# B&R Automation Studio project NewPendant_NG4_11_05_25A (part 6)

#### Main2_FourAxisTigCtrl.c.c
```c
/********************************************************************
 * COPYRIGHT -- wsi
 ********************************************************************
 * Program: Master
 * File: Master.c
 * Author: wsi
 * Created: September 25, 2012
 ********************************************************************

 Hardware[1].Inp[23] - index 80x switch
 * Implementation of program Master
 ********************************************************************/
#include <bur/plctypes.h>

#ifdef _DEFAULT_INCLUDES
#include <AsDefault.h>
#endif

#include <math.h>

#include <..\GlobDef.h>
#include <..\..\Lib\WSI_Lib.c>

#include <..\GlobDecl.h>
#include <..\Hardcoded.c>
#include <..\HMI_Cntrl.c>
#include <..\HeadConfig.c>

#include <..\..\Lib\Statelib.c>
#include <..\..\Lib\LCDLib.c>
#include <..\..\Lib\DrillMenuLib.c>
#include <..\..\Lib\LoggerLib.c>

//#include <..\..\Lib\utilityLib\bgdebug.h>
//#define TEST_ONLY_PLC_ANDROID
#define HASH_NUM				442
//#define VERSION "UnivCntrl-10-29-19B" was tested by welders
//#define VERSION "UnivCntrl-11-20-19F" // was ready for testing before Thanksgiving but nobody tested it
//#define VERSION "UnivCntrl-01-10-20F" // Successfully tested in January - very good result
//#define VERSION "UnivCntrl-02-14-20F"
//#define VERSION "UnivCntrl-02-17-20B"
//#define VERSION "UnivCntrl-02-27-20B"
//#define VERSION "UnivCntrl-03-13-20Exp"
//#define VERSION "UnivCntrl-04-17-20A" // ESTOP does not interrupt GAS
//#define VERSION "UnivCntrl-05-15-20exp" // was working
//#define VERSION "UnivCntrl-06-12-20exp"  // Max Osc ampit was changed to 3 inch
// New OSC Concept for BPV v2 is possible - make changes in Configure_BPV_v2 in OSC motor def and OSC Process use type 10
//#define VERSION "UnivCntrl-06-16-20F"  //  New Heads: BPV 2.0 MT-BO (replaces "BPV 2.0 MPBO") , BPV 2.0 TT-BO , BPV 2.0 MT-BO_TOS , BPV 2.0 TT-BO_TOS;
//BPV_v2_TT_BO_TOS chyba dziala , przenioslem w desperacji wszystko z MBPOH , trzeba dodac w Main2 wszystko zwiazane z nowymi headami
//#define VERSION "UnivCntrl-07-10-20A"
//#define VERSION "UnivCntrl-07-23-20A"
//#define VERSION "UnivCntrl-07-27-20A"
//#define VERSION "UnivCntrl-08-20-20F" // good working install on 5 machines in October 2020
//#define VERSION "UnivCntrl-09-14-20B" // new TML organization )comments) - just started
//#define VERSION "UnivCntrl-09-16-20A" // new TML organization (comments) - compiled but never used
//#define VERSION "UnivCntrl-10-27-20A" // new TML organization (comments) + SweachtHead for WF is fixed in SuperMini- is tested
//#define VERSION "UnivCntrl-11-19-20F" // the exactly the same as  "UnivCntrl-10-27-20A" but installed on Tyler machine
//#define VERSION "UnivCntrl-11-24-20F" // all as above plus file name fixed
//#define VERSION "UnivCntrl-01-29-21F" // Installed on real machine with SMH

//#define VERSION "UnivCntrl-06-04-21B" // starting - adding weld report HMI

//#define VERSION "UnivCntrl-08-09-21G" // wyjechalo do Occonee - na razie spakowane - dzialalo dobrze byli zadowloeni
//#define VERSION "UnivCntrl-08-26-21A" // proba uzycia CMT

//#define VERSION "UnivCntrl-09-02-21A" // Mode 2 nie dzialal w SuperMini ?? spowrotem Mode 1 //TVL_ROT_Param_Set[i].Mode = 2; //TVL_MODE_BPV_PosMode
// aby dzialal TVL Mode 2,3 - jazda wg position to trzeba dodac w drivie POSTRIGG2=2147483647 , POSTRIGG3=2147483647 , POSTRIGG4=2147483647
//#define VERSION "UnivCntrl-09-21-21F"
//define VERSION "MIGE_EXP-10-11-21F"
//#define VERSION "MIGE_EXP-10-13-21F"
//#define VERSION "MIGE_EXP-10-14-21G"
//#define VERSION "MIGE_EXP-10-15-21F"
//#define VERSION "MIGE_EXP-10-19-21F"
//#define VERSION "UnivCntrl-10-19-21F"
//#define VERSION "UnivCntrl-10-19-21M"
//#define VERSION "UnivCntrl-10-19-21MX"
//#define VERSION "UnivCntrl-11-02-21MX"
//#define VERSION "UnivCntrl-11-10-21MX"  // Zmiany W MIG EXP - 0.5 s delay przy restarcie pojednyczych TML
//#define VERSION "UnivCntrl-11-10-21MX"  // Zmiany W MIG EXP - 0.5 s delay przy restarcie pojednyczych TML

//#define VERSION "UnivCntrl-02-16-22A"  // dziala RUBIX

//#define VERSION "UnivCntrl-02-23-22A"  // dzial  MINI Standard

//#define VERSION "UnivCntrl-03-01-22F"  // Synch Pulse  MINI Standard & Rubix

//#define VERSION "UnivCntrl-03-24-22F"  // Poprawki w beat logger + Synch Pulse  MINI Standard & Rubix

//#define VERSION "UnivCntrl-04-05-22F"  // MiniHead Omega  +>   Poprawki w beat logger + Synch Pulse  MINI Standard & Rubix
// required -> UnivCntrl_01Apr22_US_4AXIS RUBIX & STND&MiniOmega.m.zip

//#define VERSION "UnivCntrl-04-12-22H" // poprawiony TVL step w Mode 2 i 3
// required -> UnivCntrl_01Apr22_US_4AXIS RUBIX & STND&MiniOmega.m.zip

//#define VERSION "UnivCntrl-04-29-22F" // nowy D-Head
// required -> UnivCntrl_29Apr22_US_4AXIS RUBIX & STND&MiniOmega&DHead.m.zip

//#define VERSION "UnivCntrl-06-23-22F" // nowy D-Head
// required -> UnivCntrl_21June22_US_4AXIS RUBIX & STND&MiniOmega&DHead.m.zip

// this was changed TVL_ROT_Param_Set[i].Mode = 3; to Mode 1
// in BPV_v2_MPBO head to get infinity welding
//#define VERSION "UnivCntrl-12-05-23F"
// required -> UnivCntrl_21June22_US_4AXIS RUBIX & STND&MiniOmega&DHead.m.zip

// New Head definition - BPV v2 MT  - like BPV2 but with MT truck - no position mode in TVL
//#define VERSION "UnivCntrl-12-06-23F"
// required -> UnivCntrl_21June22_US_4AXIS RUBIX & STND&MiniOmega&DHead.m.zip

//#define VERSION "UnivCntrl-12-11-23F" //New Head definition - BPV v1 MT
// required -> UnvCntrl_BPV_11_12_23.m // nowy TVL head
// required -> UnivCntrl_21June22_US_4AXIS RUBIX & STND&MiniOmega&DHead.m.zip

//#define VERSION "UnivCntrl-12-14-23F" //WYWALONY potencjometr z AVC New Head definition - BPV v1 MT
// required -> UnvCntrl_BPV_11_12_23.m // nowy TVL head
// required -> UnivCntrl_21June22_US_4AXIS RUBIX & STND&MiniOmega&DHead.m.zip

//#define VERSION "UnivCntrl-07-12-24A" // dodane BPV_v2_Video i zmiany W HMI Report

//#define VERSION "UnivCntrl-07-23-24A" // dodane BPV_v2_Video i zmiany W HMI Report

//#define VERSION "UnivCntrl-07-31-24F" // all above plus AVC feedback calibration in all legacy heads fixed

//#define VERSION "UnivCntrl-08-01-24G" // Weld Report : Heat Input or Power Ratio

//#define VERSION "UnivCntrl-09-09-24G" // Weld Report : Heat Input or Power Ratio + Limits

//#define VERSION "UnivCntrl-09-09-24R" // Radom - Weld Report : Heat Input or Power Ratio + Limits

//#define VERSION "UnivCntrl-10-18-24A" // new head : ClamShell , small change in reports

//#define VERSION "UnivCntrl-11-07-24A" // New Head KKL
//#define VERSION "UnivCntrl-11-29-24A" // New Head KKL
//#define VERSION "UnivCntrl-12-02-24A" // New Head KKL
//#define VERSION "UnivCntrl-12-03-24A" // New Head KKL

//#define VERSION "UnivCntrl-12-04-24F" // taki zostawiam przed wyjazdem
//#define VERSION "UnivCntrl-12-11-24A" // Added cherrypoint head - BP

//#define VERSION "UnivCntrl-12-30-24A" // Wire Angle Btn Fixed

/*
#ifdef MIG_SYSTEM
	#define VERSION "NG4_C15-01-14-25A" // Wire Angle Zero Btn Fixed
#else
	#ifdef CMT_SYSTEM
		#define VERSION "CMT_C15-01-14-25A"
	#else
		#define VERSION "MPC_C15-01-14-25A" // Wire Angle Zero Btn Fixed
	#endif
#endif*/

//#define VERSION "01-16-25H"  // Universal version for ClamSHell , CherryPoint & CMT , New Weld Report

//#define VERSION "01-27-25A"  // Weld Report changes - new drives cfg for ClamShell
// required -> UnvCntrl_CLAMSHELL_2025_27Jan.m

//#define VERSION "01-30-25F"  // One Wrist for BPV video Weld Report changes - new drives cfg for ClamShell ,
// required -> UnvCntrl_CLAMSHELL_2025_27Jan.m

//#define VERSION "02-03-25A"  // new head - Cherry Point BPV2 Mig Track, ++ w TVL_ROT gdy TVL continues zmiana na Mode 1
// required -> UnvCntrl_CLAMSHELL_2025_27Jan.m

//#define VERSION "02-12-25F"  // WRST TML calling fixed TML_mgr[0].hrdw[1].AxisNum = 13;
// required -> UnvCntrl_CLAMSHELL_2025_27Jan.m
//#define VERSION "02-13-25F"  // Limited list of heads
//#define VERSION "02-18-25F"  // Problem with TVL MT Mode 3 solved - Limited list of heads

// Nowy runtime , Nowe App_Config_ID i inaczej pamiec skonfigurowana
//#define VERSION "03-11-25A"  // WF & WP dziala
//#define VERSION "03-12-25A"  // AVC sense dziala
//#define VERSION "03-13-25F"  // To dzialalo i spawalo

//#define VERSION "03-13-25K"  // dodano klucz NG4_TIG_SYSTEM
//required -> UnvCntrl_CLAMSHELL_2025_27Jan.m
// required -> UnvCntrl_MIG_TIG_13Mar2025

//#define VERSION "08-01-25A"  // Nowy Pendant NG4 - proba na maszynie

//#define VERSION "08-06-25J"  // Nowy Pendant NG4 ale proba na maszynie NG4 controler

//#define VERSION "08-07-25A"  // Nowy Pendant NG4 ale proba na maszynie NG4 controler
//#define VERSION "08-07-25K"  // Nowy Pendant NG4 proba na maszynie NG4 controler _PODSTAWA do Krakowa - SPAWAL

//#define VERSION "08-11-25B"  // base for VNC pendant development

//#define VERSION "09-01-25A" // pierwsze prace w Krakowie
//#define VERSION "09-02-25A" // pierwsze prace w Krakowie
//#define VERSION "09-03-25B" // pierwsze prace w Krakowie

//#define VERSION "09-05-25A" // pierwsze prace w Krakowie
//#define VERSION "09-06-25A" // pierwsze prace w Krakowie

//#define VERSION "09-08-25A" // pierwsze prace w Krakowie
//#define VERSION "09-11-25A" // pierwsze prace w Krakowie

//#define VERSION "09-12-25A" // pierwsze prace w Krakowie

//#define VERSION "09-14-25A" // pierwsze prace w Krakowie

//#define VERSION "09-16-25A" // pierwsze prace w Krakowie
//#define VERSION "09-17-25A" // pierwsze prace w Krakowie
//#define VERSION "09-18-25A" // pierwsze prace w Krakowie
//#define VERSION "09-19-25A" // Taki przylecial z Krakowa

//#define VERSION "10-21_25A" // pierwsze uruchomienie na maszynie
//#define VERSION "10-22_25A" // proba uruchomienia tez na MPC
//#define VERSION "10-24_25D" // proba uruchomienia tez na MPC
//#define VERSION "10-30_25B" // start na CLAM SHELL maszynie
//#define VERSION "10-31_25D" // start na CLAM SHELL maszynie

//#define VERSION "11-03_25A" // start na CLAM SHELL maszynie
//#define VERSION "11-04_25A" // start na CLAM SHELL maszynie

#define VERSION "11-05_25A" // TVL Balance DIst. added

// For new pendant
_GLOBAL HARDWARE_obj hardware;
_GLOBAL MTR_obj motors[4]; // NUM_MOTORS

void FourAxisTIG();

/////////////////

_LOCAL DINT 	statusInit;

_LOCAL plcbit   MIG_ESTOP_Rst_Out , MIG_ESTOP_Rst_Btn_Inp , MIG_ESTOP_Rst_PendantBtn;

_LOCAL Cfg_typ *cfg;
_LOCAL CurCfg_typ *curCfg;
_LOCAL CurCalib_typ *curCalib, *defCalib;
_LOCAL Scaled_Var_obj *var;

_LOCAL MASTER_typ * m;
_LOCAL SerialPortDriver_typ * rs;
_LOCAL LCD_MGR_obj * lcd;
_LOCAL PENDANT_HARDWARE_obj * pend;
_LOCAL HMI_typ * hmi;
_LOCAL HMI_INTRF_typ * intrf;

_LOCAL LCD_NODE_obj * nodes;
_LOCAL TON_typ	WF_Catch_TMR;
_LOCAL UINT 	WF_RAMPUP_Comp_Step;

_LOCAL TON_typ	DoubleStop_TMR;
_LOCAL plcbit	DoubleStopBtn;
_LOCAL plcbit	DoubleStopBtn_Latch, StopBtn_Latch;

_LOCAL TON_typ	ESTOP_Dly_Tmr, AndroidConnect_Tmr;
_LOCAL UDINT	GlblBtnLED_Mask;
_LOCAL plcbit	ESTOP_PERMIT;

_LOCAL TON_typ Restart_Tmr;

//_LOCAL UINT CalibStep;
//_LOCAL BOOL CalibStepDone;
prcsSTATUS_Enum _ProcStatus;

_LOCAL INT		ANDROID_Pendant;
_LOCAL plcbit	StartBtn, StopBtn;

_LOCAL TON_typ	WireDisable_TMR;
_LOCAL UINT 	TVL_Latch_Cnt, TVL_Latch_Tm;
_LOCAL UINT 	TVL_Latch_Latched, _TVL_Latch_Latched;

_LOCAL plcbit   SYSTEM_LOCKED;

_LOCAL plcbit	Force_ENTR_LCD, _Force_ENTR_LCD;
_LOCAL UINT 	DebaunceCnt[16], DebounceTickSw, DebounceTickSwMax;
_LOCAL BOOL 	TickSw, _TickSw;
_LOCAL DINT 	WF_TVL_Diff;

INT 			_curZone;

_LOCAL plcbit	FirstScan, RefreshAndroid;

_LOCAL DINT 	_TIG_Mode , _AVC_Mode , _TVL_SYN_MODE , _WF_SYN_MODE , _WP_SYN_MODE ;

BOOL			SendRS232, _SendRS232;
_LOCAL plcstring txt[16][32];
_LOCAL Calib_Param_typ tempCalib;

_LOCAL plcbit	_segmSw;

_LOCAL plcbit	ROM_USB;

//_LOCAL DINT 	_SETUP_HEAD_SETUP;
_LOCAL plcbit	AutoStartEnable;

_LOCAL DINT 	actTicks, actTickBalance, actRot, _actRot, actPathCnt;
_LOCAL DINT 	deltaTick, actTicksForZone, actTicksForHead, actTVL_Dist, encHome_TVL;
_LOCAL DINT 	tickEncoder, _tickEncoder, encDelta;
_LOCAL UINT 	btnProgress, btnProgressMax, btnProgressBias;
_GLOBAL UINT 	curTML_indx , TML_Setup_From_Diagn;
_LOCAL UINT	    stillRun;

float			_TIG_CalibAmp, _HW_CalibAmp;

//_LOCAL Calib_Param_typ tempCalibPar;
_LOCAL UINT			_ToolHeadID , _ToolHeadID_Sw1 , _ToolHeadID_Sw2;
DINT			_GlblBtnCmd[2];

INT 			_AndroidWheel;
UINT			_AndroidEntrBtn;
_LOCAL plcstring LineTxt[256];
_LOCAL INT		parametersDump_Step, paramIndx;
_LOCAL DTStructure DTStruct;
_LOCAL DTGetTime_typ DTGetTime_1;

UDINT			_datagramCountTotal[2];
UDINT			_datagramPerSec[2];

USINT 			_MappingActive;

UINT			_PLC_Changes;
USINT 			_WireDisabled;
_LOCAL plcbit	AutoStartBtn;
_LOCAL plcbit	Cont_Stop_By_End;

_LOCAL plcbit   TIG_MIG_Sw_Inp;

_LOCAL plcbit   MIG_ESTOP_Rst_Out , MIG_ESTOP_Rst_Btn_Inp, MIG_ESTOP_Rst_Btn_Virt;
_LOCAL plcbit   Pend_Btn_Start_Virt , Pend_Btn_Stop_Virt;
_LOCAL plcbit 	MIG_Btn_Left_Inp, MIG_Btn_Right_Inp , MIG_Btn_Stop_Inp;

_LOCAL plcbit 	MIG_Btn_Left_Inp_Virt, MIG_Btn_Right_Inp_Virt ;

//_LOCAL UINT POPUP_EVENT;

_LOCAL plcbit ESTOP_Inp_Status;

_LOCAL Robot_typ * robot;

_LOCAL UINT KK_ErrorsHold;
_LOCAL UINT KK_Can_Download_Everything;

_LOCAL USINT KK_Was_Cahnged , KK_Catched;
_LOCAL USINT	KK_Life;
_LOCAL BOOL 	KK_AUTO_Test;
_LOCAL plcstring KK_text[64];
_LOCAL INT		KK_AndroidWheelIncr;
_LOCAL INT		KK_Drill, KK_Out, KK_ZONE;
_LOCAL DINT 	KK_actPosProcss , KK_ActEnc;
_LOCAL float	KK_CatchAndroidComErr;
_LOCAL UINT 	KK_CatchAndroidErr;
_LOCAL UINT 	KK_test;
_LOCAL plcbit 	KK_ClearErr;

_LOCAL USINT KK_FirstRestart_Loop;

_LOCAL DINT 	myCounter;

_LOCAL USINT   AmpsCalib_step;

_LOCAL UINT TML_Restart_Indx , TML_Restart_Step;
_LOCAL UINT Process_Restart_Indx , Process_Restart_Step;

_LOCAL float KK_ZigZag_Dist , KK_Balance_Dist;

// TVL_MAPPing
_GLOBAL DINT _deltaAPOS[TML_SERVO_NUM] , _deltaAPOS2[TML_SERVO_NUM];
_GLOBAL UINT TVL_MAP_Indx[TML_SERVO_NUM], TVL_MAP_Indx_New[TML_SERVO_NUM];
_LOCAL  UINT TVL_MAP_Step;
_LOCAL  plcbit TVL_MAP_Allowed;
void TVL_Map_ToFile();

void ProcessEvents_Android(MASTER_typ * m, LCD_NODE_obj * nodes, HMI_typ * hmi, HMI_INTRF_typ * intrf);
void EditParam(UINT paramIndx);
void JogProcessAndroid(HMI_INTRF_typ * intrf, UINT procIndx, float gain);
void TakeNextWeldProgram(HMI_typ * hmi);
void AndroidHelper(MASTER_typ * m, UINT n);

void CalibrationModePendantButtons(MASTER_typ * m, HMI_typ * hmi, HMI_INTRF_typ * intrf, LCD_MGR_obj * lcd);
void StopModeAndroidButtons(MASTER_typ * m, HMI_typ * hmi, HMI_INTRF_typ * intrf, LCD_MGR_obj * lcd);
void StopCalibrationModeAndroidButtons(MASTER_typ * m, HMI_typ * hmi, HMI_INTRF_typ * intrf, LCD_MGR_obj * lcd);
void RunModeAndroidButtons(MASTER_typ * m, HMI_typ * hmi, HMI_INTRF_typ * intrf, LCD_MGR_obj * lcd);
void RunCalibrationModeAndroidButtons(MASTER_typ * m, HMI_typ * hmi, HMI_INTRF_typ * intrf, LCD_MGR_obj * lcd);

DINT MasterSequence(MASTER_typ * m, HMI_typ * hmi, plcbit StartBtn, plcbit StopBtn);
DINT MasterSequence_Contin(MASTER_typ * m, HMI_typ * hmi, plcbit StartBtn, plcbit StopBtn);
DINT MasterSequence_Contin_OneWay(MASTER_typ * m, HMI_typ * hmi, plcbit StartBtn, plcbit StopBtn);

DINT CalibrationSequence(MASTER_typ * m, HMI_typ * hmi, plcbit StartBtn, plcbit StopBtn);

void IncrParam(CurCfg_typ * curCfg, UINT param, DINT segm, float gain);
void DecrParam(CurCfg_typ * curCfg, UINT param, DINT segm, float gain);

void Check_parOSC_Excur(CurCfg_typ * curCfg, HMI_typ * hmi, UINT seg);

void Check_parOSC_Amplit(CurCfg_typ * curCfg, HMI_typ * hmi, UINT seg);
void PleaseUpdateHeadSetup(MASTER_typ * m);

void SetBannerTxt(MASTER_typ * m, HMI_typ * hmi, HMI_INTRF_typ * intrf);
float getBtnProgress();
void SetZeroPosition(MASTER_typ * m);
void CreateParamList();
void DeleteExtension(char * p);
void WireDisableInable(plcbit Tmr_Q);

void DumpParamToFile();
void EvaluatePosition();
void Fill_Segments(CurCfg_typ * curCfg, UINT par, UINT seg, UINT Mode, UINT Step);

int WatchArcLinkError(MASTER_typ * m, Robot_typ * robot);
DINT Check_OSC_Amplt_and_Center();

void CalculateRunOverlap();
void CalculateRunOverlap_Cont();
void CalculateRunOverlap_Cont_OneWay();

void RestartStateMach();
plcbit Find_ext_txt(char *name , char* ext);

_LOCAL DINT _NextHeadConfig_Indx;

void _INIT Main2_INIT(void)
{
UINT i;

	KK_ZigZag_Dist = 20;

	//////////////////////////////////
		// Pozostalosci po SuperMaster
		// do przeanalizowania
	#ifdef  MIG_SYSTEM

		ProjectConfig_Hrdw = project_FourAxisTig;
		ProjectConfig = project_FourAxisTig;

	#endif
		FourAxisTIG();

	///////////////////////////////////

#ifdef MIG_SYSTEM
	strcpy(PLC_Version_TXT, "NG4-"); //#define VERSION "NG4_C15-01-14-25A" // Wire Angle Zero Btn Fixed
#else
	#ifdef CMT_SYSTEM
	strcpy(PLC_Version_TXT, "CMT-");
	#else
	strcpy(PLC_Version_TXT, "MPC-");
	#endif
#endif

	strcat(PLC_Version_TXT, VERSION);

#ifdef CHERRYPOINT_LIST

	strcat(PLC_Version_TXT, "-CP");

#endif

	LimScal_Tilt.x1 = 0.0;
	LimScal_Tilt.y1 = 0.0;

	LimScal_Tilt.x1 = 4096.0;
	LimScal_Tilt.y1 = 360.0;

	//	Program options
	KK_DoNotChangeTMLProgram 	= 0;
	KK_DoNotHashCalculation 	= 1; // always like that
	TVL_MAP_Allowed 			= 0;
	KK_No_TVL_Restart	= 0;
	KK_ManualCalib		= 0;
	KK_TML_PowerON		= 0;
	KK_Functionality	= 0;
	KK_ErrorsHold 		= 0;
	KK_Can_Download_Everything = 0;

	//////////////////////////
	Hold_Estop_ON 		= 0;
	ESTOP_Inp_Status 	= 0;
	TVL_Latch_Tm		= 50;
	ANDROID_Pendant 	= 1;

	//some heads setup in Config
	btnProgressMax		= 50;
	btnProgressBias 	= 10;

	KK_AUTO_Test		= 0;

	DebounceTickSwMax	= 2;

	// Just to see globals in the watch window
	Master[0].Active	= Master[0].Active;

	//LCD_MGR[0].curHead = LCD_MGR[0].curHead;
	RS232[0].Ident		= RS232[0].Ident;
	Pendant[0].ABEncoder = Pendant[0].ABEncoder;

	ESTOP_Dly_Tmr.PT	= 1000; 					// 1 sec delay off ESTOP
	Hardware[0].Inp[4]	= 1;						// ESTOP

	Master[0].AndIntrf[0].Alive = 0;

	myCounter			= myCounter;

	ReadPermMemory_HS.Go = 0;
	ReadPermMemory_HS.Ready = 0;

	ReadCfgFile_HS.Go = 0;
	ReadCfgFile_HS.Ready = 0;

	TimerStart(&DoubleStop_TMR, 1.0);
	TimerExecute(&DoubleStop_TMR);

	Hardware[1].Outp[9] = 0; // Lights OFF (NC) on camera

	FirstScan = 1;
	RefreshAndroid = 0;

	SYSTEM_LOCKED = 0;

	LoggerInit(&LogMgr, &LogID, "LogBook1", 2000);

	// Very Important - get value from Statis Memory
	_NextHeadConfig_Indx = NextHeadConfig_Indx;
	actTicks			= actTicksPerm;

	if((_NextHeadConfig_Indx < 0) || (_NextHeadConfig_Indx >= HEAD_INVALID)){
		_NextHeadConfig_Indx = BPV_v2;
		NextHeadConfig_Indx = BPV_v2;
	}

	Master[0].ToolHeadID = (UINT)LastHeadDir;

	for(i = 0; i < HEAD_INVALID ; i++)
		AssignHeadText(NewHeadName[i] , i);

	strcpy(curHeadName , NewHeadName[NextHeadConfig_Indx]);

}

void _CYCLIC Main2_CYCLIC(void)
{
int 			i, k;
char			status, _status;
DINT			d;
int 			len;
float 			x;

//plcbit StartBtn , StopBtn;
INT 			tickIncr;
LCD_NODE_obj *	curNode;

	#ifdef MIG_PENDANT

		m		= pMaster[1];
		lcd 	= pLCD_MGR[1];
		rs		= pRS232[1];
		pend	= pPendant[1];

	#else

		m		= pMaster[0];
		lcd 	= pLCD_MGR[0];
		rs		= pRS232[0];
		pend	= pPendant[0];

	#endif

	if(SYSTEM_LOCKED) // System Locked after Head definition changed - Must reboot
		return;

	// Check if pointers are not null
	if (!m)
		return;

	nodes				= m->pNode[0];

	if (!nodes)
		return;

	if (!lcd)
		return;

	if (!rs)
		return;

	if (!pend)
		return;

	if (!m->pCurCfg || !m->pCfg || !m->pCalib || !m->pScaledVar)
		return;

	cfg 				= (Cfg_typ *)		m->pCfg;
	curCfg				= (CurCfg_typ *)	m->pCurCfg;
	curCalib			= (CurCalib_typ *)	m->pCalib;
	defCalib			= (CurCalib_typ *)	m->pDefaultCalib;
	var 				= (Scaled_Var_obj*)	m->pScaledVar;
	robot				= (Robot_typ*)PS_Param_Set[0].pArcLinkRobot;

	hmi 				= &m->Hmi[0];
	intrf				= &m->Intrf[0];

	if (!hmi || !intrf)
		return;

	////////////////////////////////////////

	if(KK_ClearErr){
		KK_ClearErr = 0;
		KK_AckAllErrors(&ErrorMgr);
	}
	//////////////////////////////////////

	Hardware[1].Outp[8] = Hardware[1].Outp[9]; // Power on Camera #1

	///////// Important because HMI in Global setting can change NextHeadConfig_Indx

	// Head type was changed - Load New Head definition

	if(hmi->curHeadID != P_PARAM_GLOBAL){

		if(_NextHeadConfig_Indx != NextHeadConfig_Indx){
			_NextHeadConfig_Indx = NextHeadConfig_Indx;

			LogTxt(&LogMgr, "Head was changed");

			/*
			STOP_SavingData = 1;
			m->sm.Step = 1001;
			m->LOCKED = 1;
			TML_MTR_CUT_POWER = 1;
			*/

			FirstScan = 1;

			#ifdef  MIG_PENDANT

			m->sm.Step = 1;

			#else

			RefreshAndroid = 1;
			TML_MTR_CUT_POWER = 1;

			m->LOCKED = 1;
			m->sm.Step = 250;

			#endif

		}

	}

	if(FirstScan){
		FirstScan = 0;

		ReadPermMemory_HS.Ready = 0;
		ReadPermMemory_HS.Go = 1;
		m->xCmd = mstrRESTART;

		LogTxt(&LogMgr, "System Restart");

	}

	//////////////////////////////////////////////////////////////////
	DumpParamToFile();

	if(TVL_MAP_Allowed)
		TVL_Map_ToFile();

	////////////////////////////////////////////////////
	// Task restart from supemaster
	if ((m->xCmd == mstrRESTART))
	{

		if(m->pNode[0] && ReadPermMemory_HS.Ready)
		{

			sm_init(&m->sm);
			pend->_intr.TickIncr = 2;

			for (i = 0; i < PROCESS_NUM; i++)
				Process[i].ConfigReady = 0;

			//SerialPortInit(rs ,  pend->RSDeviceStr , "/PHY=RS232 /BD=9600 /DB=8 /PA=N /SB=1");
			//SerialPortInit(rs , "IF1" , "/PHY=RS232 /BD=9600 /DB=8 /PA=N /SB=1");
			SerialPortInit(rs, "IF6.ST11.IF1", "/PHY=RS232 /BD=9600 /DB=8 /PA=N /SB=1");

			//SerialPortInit(rs , "SS1.IF1.ST5.IF1.ST4.IF1" , "/PHY=RS232 /BD=9600 /DB=8 /PA=N /SB=1");

			/** Master reinit **/
			m->varLastNum		= varLAST_VARIABLE;
			m->paramLastNum 	= parLAST_PARAM;
			m->numSegm			= SEGM_NUM_MAX;
			m->paramEnumLastNum = parENUM_LAST_PARAM;
			m->varEnumLastNum	= varENUM_LAST_VARIABLE;
			m->paramIntgLastNum = parINT_LAST_PARAM;
			m->varIntLastNum	= varINT_LAST_VARIABLE;
			m->paramStrLastNum	= parSTRING_LAST_PARAM;
			m->varStrLastNum	= varSTRING_LAST_VARIABLE;

			memset(nodes, 0, sizeof(LCD_NODE_obj) *NODES_NUM_MAX);

			//ScaledValuesCfg(m); // This is pointer population
			HardCodeCFg(m); 						// This is for pamaeters and variable definition

			#ifdef MIG_PENDANT

			for (i = 0 ; i < m->paramLastNum; i++){

				//curCfg->Param[i].segmYes = cfg->Param[i].SegmType;
				if(cfg->ScaledVar[i].segm == 1)
					curCfg->Param[i].segmYes = 1;
				else
					curCfg->Param[i].segmYes = 0;

			}

			#endif

			CreateParamList();

			SetupNODES_Android(m, nodes, P_LAST_NODE); // this is what will be displayed on LCD - menu etc

			statusInit			= LCD_MGR_Init(lcd, NUM_LINE, NODES_NUM_MAX, m, rs, nodes, P_INIT, 0.05);

			lcd->EditMode		= EDIT_MODE_VALUE;	// Edit only value of parameter on the screen

			//////////////////////////////////////////
			// Assign HMI pointers from external instances
			for (i = 0; i < 20; i++)
				hmi->pHMI_Lines[i] = HMI_lines[i];

			#ifdef MIG_PENDANT

				for (i = 0; i < 4; i++)
					hmi->pMessage[i] = DrillDwnHMI.Message[i];

			#else

				for (i = 0; i < 4; i++)
				hmi->pMessage[i] = m->AndIntrf[0].Message[i];

			#endif

			hmi->pBanner		= m->AndIntrf[0].Banner;

			/////////////////////////////////////////
			TimerStart(&hmi->MsgTmr, 0.1);

			if(NextHeadConfig_Indx < U_BEND_HP_ENC)
				NextHeadConfig_Indx  = U_BEND_HP_ENC;

			if(NextHeadConfig_Indx >= HEAD_INVALID)
				NextHeadConfig_Indx= HEAD_INVALID-1;

			///////////////////////////////

			if((strlen(curCfg->NextProgramName) > 31)
				|| (strlen(curCfg->NextProgramName) == 0))
				strcpy(curCfg->NextProgramName, PRG_NO_NEXT);

			///////////////////////////////

			if(ConfigureHead(m, NextHeadConfig_Indx))
			{
				curCalib->GenSetup[SETUP_HEAD_SETUP] = NextHeadConfig_Indx;
				m->xCmd 	= 0;

				if(RefreshAndroid)
					hmi->PLC_Changes = 0x0001; // new curcCfg Loaded

				RefreshAndroid = 0;

				///// pointers to main objects so Cfg file parser can see them //
				m->Objects.pArcLink_IP_Address = (UDINT)ArcLinkPS_IP_Address;

				for(i = 0 ; i < TIG_PS_NUM ; i++)
					m->Objects.pPS_Param_Set[i] = &PS_Param_Set[i];

				///////
				_TIG_Mode = 0xFFFF;
				_AVC_Mode = 0xFFFF;
				m->Active			= 1;	// Master active
				m->sm.Step			= 0;	// Main state machine reset
				///////////////
				//ReadPermMemory_HS.Go = 1; //plus Parse Cfg File
				STOP_SavingData = 0;

				switch(curCalib->GenSetup[SETUP_HEAD_SETUP]){

					case BPV_F_HEAD:
					case BPV_v1_MT:
					case CLAMSHELL_HEAD:
					case CHERRYPOINT_BP1_HEAD:
					case CHERRYPOINT_BP2_HEAD:
					case CHERRYPOINT_MT_BP2_HEAD:
					case MIG_TIG_HEAD:

					 	DC_Mtr[m->pCfg->HeadCfg.INDX.DC_A_Indx].msc.Pos = OLD_MTR_POS[INDX_A_LAST_POS];
						DC_Mtr[m->pCfg->HeadCfg.INDX.DC_B_Indx].msc.Pos = OLD_MTR_POS[INDX_B_LAST_POS];

					break;

					case RUBIX:

						btnProgressMax		= 30;
						btnProgressBias 	= 30;

					break;

				}

				LCD_Init_Step = 0;

			}

			ESTOP_PERMIT		= 1;

			///////////////////////////////////////////
			//GB: calculate hash value for the NODES array
			if (KK_DoNotHashCalculation)
			{

				gHashValuesArray[0] = HASH_NUM;
				gHashValuesArray[1] = gHashValuesArray[0];

			}
			else
			{

				gHashValuesArray[0] = hash_of_binary_array(nodes, sizeof(LCD_NODE_obj) *NODES_NUM_MAX);
				gHashValuesArray[1] = hash_of_binary_array(cfg, sizeof(Cfg_typ));

			}

			///////////////////////////////////////////
			VectorStateMach[m->pCfg->HeadCfg.TVL.VECT_Indx].OutVect.softLimits[0] = 0.0;
			VectorStateMach[m->pCfg->HeadCfg.TVL.VECT_Indx].OutVect.softLimits[1] = 0.0;
			////////////////////////////////////////////
			TML_MTR_INST[m->pCfg->HeadCfg.AVC.TML_A_Indx]._cfg.signFilter = curCfg->Param[parAVC_FbkFilter].val[0];
			TML_MTR_INST[m->pCfg->HeadCfg.AVC.TML_A_Indx]._cfg.kpp = (DINT)(curCfg->Param[parAVC_KPP].val[0] *TML_MTR_INST[m->pCfg->HeadCfg.AVC.TML_A_Indx]._cfg.kppMax) ;
			TML_MTR_INST[m->pCfg->HeadCfg.AVC.TML_A_Indx]._cfg.kip = (DINT)(curCfg->Param[parAVC_KIP].val[0] *TML_MTR_INST[m->pCfg->HeadCfg.AVC.TML_A_Indx]._cfg.kipMax) ;

			TML_MTR_INST[m->pCfg->HeadCfg.AVC.TML_B_Indx]._cfg.signFilter = curCfg->Param[parAVC_FbkFilter].val[0];
			TML_MTR_INST[m->pCfg->HeadCfg.AVC.TML_B_Indx]._cfg.kpp = (DINT)(curCfg->Param[parAVC_KPP].val[0] *TML_MTR_INST[m->pCfg->HeadCfg.AVC.TML_A_Indx]._cfg.kppMax) ;
			TML_MTR_INST[m->pCfg->HeadCfg.AVC.TML_B_Indx]._cfg.kip = (DINT)(curCfg->Param[parAVC_KIP].val[0] *TML_MTR_INST[m->pCfg->HeadCfg.AVC.TML_A_Indx]._cfg.kipMax) ;

			for (i = 0; i < TML_SERVO_NUM; i++)
				TML_MTR_INST[i].xCMD = TML_RESTART;

			for (i = 0; i < PROCESS_NUM; i++)
				Process[i].xCMD = prcsRESTART;

			intrf->TestMode 	= 1;
			m->WireDisabled 	= 1;

		}

	}
/*
#ifndef  MIG_EXP_SYSTEM

	#ifndef CLAMSHELL

		if(!Hardware[1].CouplerOK[0]){
			Errors(&ErrorMgr,ERROR_HARDWARE, ERROR_MODULE_ERR ,1);
		}
	#endif

	#ifndef CHERRYPOINT

		if(!Hardware[1].CouplerOK[0]){
			Errors(&ErrorMgr,ERROR_HARDWARE, ERROR_MODULE_ERR ,1);
		}
	#endif

#endif
*/

#ifdef  MIG_SYSTEM

/*

	#ifndef CLAMSHELL

	if(!TIG_MIG_Sw_Inp)
		Errors(&ErrorMgr, ERROR_HARDWARE, ERROR_TIG_MIG_SW_ERR, 0);

	#endif

	#ifndef CHERRYPOINT

		if(!TIG_MIG_Sw_Inp)
			Errors(&ErrorMgr, ERROR_HARDWARE, ERROR_TIG_MIG_SW_ERR, 0);

	#endif
*/

	#ifdef MIG_PENDANT

			Pend_Btn_Stop = MIG_Btn_Stop_Inp || Pend_Btn_Stop_Virt;

			#ifdef SYSTEM_SIMULATION

			Pend_Btn_Left = MIG_Btn_Left_Inp || MIG_Btn_Left_Inp_Virt;
			Pend_Btn_Right = MIG_Btn_Right_Inp || MIG_Btn_Right_Inp_Virt;

			#else

			Pend_Btn_Left = MIG_Btn_Left_Inp;
			Pend_Btn_Right = MIG_Btn_Right_Inp;

			#endif

			Pend_Btn_Start = Pend_Btn_Start_Virt;

	#endif

	if(m->sm.Step != 191)
		MIG_ESTOP_Rst_Btn_Virt = 0;

	MIG_ESTOP_Rst_PendantBtn = (intrf->GlblBtnCmd[0] &ANDR_BTN_STOP) && Master[0].ESTOP;

	MIG_ESTOP_Rst_Out = MIG_ESTOP_Rst_Btn_Inp || MIG_ESTOP_Rst_Btn_Virt
		|| Pend_Btn_Stop;

	//MIG_ESTOP_Rst_Out = MIG_ESTOP_Rst_Btn_Inp || MIG_ESTOP_Rst_PendantBtn;

#else

	if(!Hardware[1].CouplerOK[0]){
			Errors(&ErrorMgr,ERROR_HARDWARE, ERROR_MODULE_ERR ,1);
	}

#endif

	if(ProjectConfig_Hrdw_ERROR){
		Errors(&ErrorMgr, ERROR_SETUP, ERROR_PROJECT_HRDW_ERR, 0);
	}

	/////////////////////////////////////////////////////

	EvaluatePosition();

	//////////////////////////
	// Special trick

	if((intrf->GlblBtnCmd[0] & ANDR_BTN_HOME) &&  (intrf->GlblBtnCmd[0] & ANDR_BTN_START)
		&&  (intrf->GlblBtnCmd[0] & ANDR_BTN_AVC_LOCK))
		KK_Functionality = 1;

	if((intrf->GlblBtnCmd[0] & ANDR_BTN_HOME) &&  (intrf->GlblBtnCmd[0] & ANDR_BTN_STOP))
		KK_Functionality = 0;

	//////////////////////////
	// Trigger ESTOP when TML error
	if (KK_TML_PowerON || Hold_Estop_ON){

		Hardware[1].Outp[7] = 1; // Four AXIS start Inable and Power to TML motors

		if(m->pESTOP_Out)
			*m->pESTOP_Out = 1;

	}
	else {

		Hardware[1].Outp[7] = !TML_MTR_CUT_POWER; // Four AXIS start Inable and Power to TML motors

		if(m->pESTOP_Out)
			*m->pESTOP_Out = !TML_MTR_CUT_POWER;
	}

	if (curCfg->Param[parLCD_BtnMode].val[0] > 0.0)
		lcd->EntrBtnPressReq = 1; // LCD ENtr button should be hold to edit
	else
		lcd->EntrBtnPressReq = 0;

	// UWAGA NJAWAZNIEJSZE!!!!!!!
	///intrf->GlblBtnCmd[0] = (m->AndIntrf[0].GlblBtnCmd[0] &0xFFFFFFFE); // first bit is wheel is not pressed so we mask it;

	#ifdef MIG_PENDANT

		intrf->GlblBtnCmd[0] = (HMI_Intr.GlblBtnCmd[0] & 0xFFFFFFFE);
		m->AndIntrf[0].Wheel = HMI_Intr.Wheel;

		DrillDwnHMI.StartBtn_Vis = 1; //INVISIBLE;
		DrillDwnHMI.StopBtn_Vis = 1; //INVISIBLE;
	#else

		intrf->GlblBtnCmd[0] = (m->AndIntrf[0].GlblBtnCmd[0] &0xFFFFFFFE); // first bit is wheel is not pressed so we mask it;

	#endif

	if (intrf->GlblBtnCmd[0] == 0)
		btnProgress = 0;

	intrf->Wheel		= m->AndIntrf[0].Wheel;

	intrf->WheelDelta	= m->AndIntrf[0].Wheel - _AndroidWheel;
	_AndroidWheel		= m->AndIntrf[0].Wheel;

	intrf->LCDEntr		= (m->AndIntrf[0].EntrBtn > 0);
	intrf->TickPlus 	= ((intrf->WheelDelta > 0) || ((intrf->GlblBtnCmd[0] &ANDR_BTN_UP) &&
		 !intrf->_intr._GlblBtnCmd[0]));
	intrf->TickMinus	= ((intrf->WheelDelta < 0) || ((intrf->GlblBtnCmd[0] &ANDR_BTN_DOWN) &&
		 !intrf->_intr._GlblBtnCmd[0]));

	intrf->LCDEntr_PosEdge = (m->AndIntrf[0].EntrBtn && !_AndroidEntrBtn);
	intrf->LCDEntr_NegEdge = (!m->AndIntrf[0].EntrBtn && _AndroidEntrBtn);
	_AndroidEntrBtn 	= m->AndIntrf[0].EntrBtn;

	m->AndIntrf[0].GlblBtnLED[0] = intrf->GlblBtnLED[0];

	if(intrf->TickPlus)
		myCounter++;

	////////////////////////////////////////
#ifndef MIG_PENDANT
	hmi->curHeadID		= m->AndIntrf[0].curHeadID;
	hmi->curNodeID		= m->AndIntrf[0].curLineID;

	hmi->FiredEvent 	= m->AndIntrf[0].FiredEvent;
	//hmi->PleaseUpdate	= m->AndIntrf[0].PleaseUpdate;
	hmi->UserLevel		= m->AndIntrf[0].UserLevel;
	m->AndIntrf[0].FiredEvent = 0;

#endif

	/////////////////////////////////////////
	// Security for edit on node
	if (hmi->curHeadID < P_LAST_NODE)
	{ // on one of drill down page

		if (hmi->UserLevel < nodes[hmi->curNodeID].MinUserLevel)
			intrf->LCDEntr = 0;

	}

	//////////////////////////////////////////////

	// Special Setup for particular Heads

	switch(curCalib->GenSetup[SETUP_HEAD_SETUP]){

		case BPV_v2:
		case BPV_v2_MPBO:
		case BPV_v2_MPGH:
		case BPV_v2_MPGV:

		case BPV_v2_TT_BO:
		case BPV_v2_MT_BO:
		case BPV_v2_MT_BO_TOS:
		case BPV_v2_TT_BO_TOS:
		// dodane 8July24
		case BPV_v2_Video:

		// Dodane 12Dec23
		case BPV_v2_MT:

			WRST_TML_Param_Set[0].MappingActive = (curCalib->GenSetup[SETUP_MAPPING_ON] > 0)? 1:0;

		break;

		default:

			curCalib->GenSetup[SETUP_MAPPING_ON] = 0;

			WRST_TML_Param_Set[0].MappingActive = 0;

		break;

	}

	///////////////////////////////////////////////

	switch(curCalib->GenSetup[SETUP_HEAD_SETUP]){

		case CLAMSHELL_HEAD:
		case CHERRYPOINT_BP1_HEAD:
		case CHERRYPOINT_BP2_HEAD:
		case CHERRYPOINT_MT_BP2_HEAD:
		case MIG_TIG_HEAD:
		case  BPV_v2_Video:

			if(TVL_ROT_Param_Set[0].TotalRescaleFactor != 0.0)	{

				/*
				LimScal_Tilt.x = (float)TML_MTR_INST[TML_AX_AVC].AnInp[1];
				AzzLimScal(&LimScal_Tilt);
				x = LimScal_Tilt.y - curCalib->GenFloatValue[SETUP_FLOAT_TILT_OFFSET];
				*/

				//xsprintf(m->AndIntrf[0].MasterModTXT, "Tilt:%1.1f  %d/%d TVL:%d / Enc:%d " ,x  , File_RW._int.PathDoneCnt,
										//(UINT) curCfg->Param[parGEN_WeldProgramRepeat].val[0], TVL_ROT_Param_Set[0].EncPos_FBK, actTicks);

				//xsprintf(m->AndIntrf[0].MasterModTXT, "T:%1.1f W:%1.1f  %d/%d TVL:%d / Enc:%d " ,x , TML_MTR_INST[TML_AX_WRST].PosFBK , File_RW._int.PathDoneCnt,
					 	//(UINT) curCfg->Param[parGEN_WeldProgramRepeat].val[0], TVL_ROT_Param_Set[0].EncPos_FBK, actTicks);

				xsprintf(m->AndIntrf[0].MasterModTXT, "WA:%1.1f	%d/%d TVL:%d / Enc:%d "  , TML_MTR_INST[m->pCfg->HeadCfg.WRST.TML_A_Indx].PosFBK , File_RW._int.PathDoneCnt,
						(UINT) curCfg->Param[parGEN_WeldProgramRepeat].val[0], TVL_ROT_Param_Set[0].EncPos_FBK, actTicks);

			}

		break;

		default:

			if(TVL_ROT_Param_Set[0].TotalRescaleFactor != 0.0)	{

				if(WRST_TML_Param_Set[0].MappingActive){
					//xsprintf(m->AndIntrf[0].MasterModTXT, "A:%2.1f/%2.1f / TVL:%d / Enc:%d / I:%3.2f ", 1.0/TVL_ROT_Param_Set[0].TotalRescaleFactor, WRST_TML_Param_Set[0].actAngleFromMapping,
					//xsprintf(m->AndIntrf[0].MasterModTXT, "A:%2.1f/%2.1f / TVL:%d / Enc:%d / I:%3.2f ",WRST_TML_Param_Set[0].actAngle , WRST_TML_Param_Set[0].actAngleFromMapping,
					 //TVL_ROT_Param_Set[0].EncPos_FBK, actTicks,VectorStateMach[m->pCfg->HeadCfg.INDX.VECT_A_Indx].FbkVect.x - VectorStateMach[m->pCfg->HeadCfg.INDX.VECT_B_Indx].FbkVect.x );
					xsprintf(m->AndIntrf[0].MasterModTXT, "A:%2.1f/%2.1f / TVL:%d / Enc:%d/ %d;%d  ",WRST_TML_Param_Set[0].actAngle , WRST_TML_Param_Set[0].actAngleFromMapping,
					 TVL_ROT_Param_Set[0].EncPos_FBK, actTicks,File_RW._int.PathDoneCnt, (UINT) curCfg->Param[parGEN_WeldProgramRepeat].val[0]);

				}else{

					switch(curCalib->GenSetup[SETUP_INDX_ENBL]) {

					case 1:

						xsprintf(m->AndIntrf[0].MasterModTXT, "%3.2f %d/%d TVL:%d / Enc:%d / I:%3.2f ", 1.0/TVL_ROT_Param_Set[0].TotalRescaleFactor ,File_RW._int.PathDoneCnt,
					 	(UINT) curCfg->Param[parGEN_WeldProgramRepeat].val[0], TVL_ROT_Param_Set[0].EncPos_FBK, actTicks,VectorStateMach[m->pCfg->HeadCfg.INDX.VECT_A_Indx].FbkVect.x - VectorStateMach[m->pCfg->HeadCfg.INDX.VECT_B_Indx].FbkVect.x );

					break;

					default:

						xsprintf(m->AndIntrf[0].MasterModTXT, "%3.2f %d/%d TVL:%d / Enc:%d ", 1.0/TVL_ROT_Param_Set[0].TotalRescaleFactor ,File_RW._int.PathDoneCnt,
					 	(UINT) curCfg->Param[parGEN_WeldProgramRepeat].val[0], TVL_ROT_Param_Set[0].EncPos_FBK, actTicks);

					break;

					}
				}
			}

		break;

	}

	if(curCfg->Param[parTVL_ZigZagDist].val[0] != 0.0){

		if(curCalib->GenSetup[SETUP_ZIG_ZAG])
			strcat(m->AndIntrf[0].MasterModTXT , ">");

	}

	/////////////////////////////////

#ifndef MIG_PENDANT

	EvaluateHMI_Android(m, nodes, hmi, intrf);

#endif

	 ProcessEvents_Android(m, nodes, hmi, intrf);

////////////////////////////////////////////////////////////
	 // m->curSegm[FR_SEGM]

	m->AndIntrf[0].MsgTmr_Done = !hmi->MsgTmr.Q;
	m->AndIntrf[0].MsgTmr_Duration = (UINT) (hmi->MsgTmr.PT / 1000.0);
	m->AndIntrf[0].MasterMode = m->Mode;

	if((hmi->curHeadID != P_PARAM_TIG)
		&& (hmi->curHeadID != P_PARAM_AVC)
		&& (hmi->curHeadID != P_PARAM))
		ChangeSegmentList();

	if (_PLC_Changes != hmi->PLC_Changes)
	{ // New flag
		m->AndIntrf[0].PLC_Changes = hmi->PLC_Changes; // New flag,
		_PLC_Changes		= hmi->PLC_Changes;

	}

	else if (m->AndIntrf[0].PLC_Changes == 0)
	{ // Changes accepted
		hmi->PLC_Changes	= 0;
		_PLC_Changes		= hmi->PLC_Changes;

	}

	if (!m->AndIntrf[0].xCMD)
	{

		if ((hmi->Node2JumpID >= P_MENU) && hmi->xCMD)
		{

			m->AndIntrf[0].xCMD = hmi->xCMD;
			m->AndIntrf[0].JumpLineID = hmi->JumpLineID;
			m->AndIntrf[0].Node2JumpID = hmi->Node2JumpID;

			#ifndef MIG_PENDANT
			hmi->xCMD			= 0;
			hmi->JumpLineID 	= 0;
			hmi->Node2JumpID	= 0;
			#endif
		}
		else
		{
			if(hmi->xCMD){
				m->AndIntrf[0].xCMD = hmi->xCMD;

				#ifndef MIG_PENDANT
				hmi->xCMD = 0;
				#endif
			}
		}
	}

	// No Buttons pressed when pop up message is on
	// I removed it because I could not evaluate holding buttons - 8 November 2017
	/*
	if (m->AndIntrf[0].MsgTmr_Done)
	{
		intrf->GlblBtnCmd[0] = 0;
		m->AndIntrf[0].GlblBtnCmd[0] = 0;
	}
	*/

	///////////////////
	// Buttons
	m->AndIntrf[0].GlblBtnLED[0] = 0;

	if (intrf->TestMode)
		m->AndIntrf[0].GlblBtnLED[0] |= 0x1;

	if (!m->WireDisabled)
		m->AndIntrf[0].GlblBtnLED[0] |= 0x2;

	if (Process[m->pCfg->HeadCfg.AVC.PROC_Indx].Param[0])
		m->AndIntrf[0].GlblBtnLED[0] |= 0x4;

	if (Process[m->pCfg->HeadCfg.GAS.PROC_Indx].Status != prcsSTATUS_Stopped)
		m->AndIntrf[0].GlblBtnLED[0] |= 0x8;

	if (!m->ToolHeadID)
		m->AndIntrf[0].GlblBtnLED[0] |= 0x10;
	else
		m->AndIntrf[0].GlblBtnLED[0] |= 0x20;

	m->AndIntrf[0].GlblBtnLED[1] = 0;

	switch (curCalib->GenSetup[SETUP_OSC_EXC_MODE])
	{
		case 1:
			m->AndIntrf[0].GlblBtnLED[1] |= 0x1;
			break; // Dwell In

		case 2:
			m->AndIntrf[0].GlblBtnLED[1] |= 0x2;
			break; // Dwell Out

		default:
			break; // Excursion time
	}

	//m->AndIntrf[0].curNumSegments = m->numZone;
	//m->AndIntrf[0].maxNumSegments = FR_SEGM_NUM_MAX;
	m->AndIntrf[0].curNumSegments = m->curSegm[ZONE];
	m->AndIntrf[0].maxNumSegments = m->numZone + 1;

	Master_numZone = m->numZone;

	hmi->xCMD = 0;

	/********************************************************/

	if (m->ESTOP && lcd->Intr.SlowBlink)
		strcpy(lcd->Banner, "	ESTOP !!!!! ");

	if (Force_ENTR_LCD)
	{
		intrf->LCDEntr		= 1;
		lcd->EditMode		= EDIT_MODE_VALUE;
		lcd->Intr.editStep	= 3;
	}

	if (Force_ENTR_LCD && !_Force_ENTR_LCD)
		intrf->LCDEntr_PosEdge = 1;

	else if (!Force_ENTR_LCD && _Force_ENTR_LCD)
		intrf->LCDEntr_NegEdge = 1;

	_Force_ENTR_LCD 	= Force_ENTR_LCD;

	Force_ENTR_LCD		= 0;

	if (!ANDROID_Pendant)
	{

		if (statusInit == 1)
		{

			lcd->Intrf.WheelDelta = intrf->WheelDelta;

			lcd->Intrf.LCDEntr	= intrf->LCDEntr;
			lcd->Intrf.LCDEntr_NegEdge = intrf->LCDEntr_NegEdge;
			lcd->Intrf.LCDEntr_PosEdge = intrf->LCDEntr_PosEdge;

			lcd->Intrf.TickMinus = intrf->TickMinus;
			lcd->Intrf.TickPlus = intrf->TickPlus;

			status				= LCD_MGR_Srv(lcd);

			// Trigger sending to screen every second loop
			if (SendRS232)
			{

				if (!rs->txBufRequest)
					rs->txBufRequest = 1;

			}

			SendRS232			= !SendRS232;
			/****************************************/
		}
	}

	/************************************************************/

	if (m->LOCKED && (m->sm.Step < 230))
	{

		for (i = 0; i < PROCESS_NUM; i++)
			Process[i].xCMD = prcsHalt;

		for (i = 0; i < TML_SERVO_NUM; i++)
			TML_MTR_INST[i].xCMD = TML_RESET_ONLY_CMD;

		m->Mode 			= MASTER_MODE_INIT;

		STOP_SavingData = 1;
		m->sm.Step			= 230;
	}

	////////////////////
	// Android connection
	if (ANDROID_Pendant)
	{

		if ((m->sm.Step > 1))
		{ // Allow init first

			if (_datagramCountTotal[0] != datagramCountTotal[0])
				TimerStart(&AndroidConnect_Tmr, 1.5);
				//TimerStart(&AndroidConnect_Tmr, 1.0);

			if (TimerIsTimeOut(&AndroidConnect_Tmr))
			{

				AndroidConnect_Tmr.IN = 0;
				AndroidConnect_Tmr.Q = 0;

				if (m->AndIntrf[0].Alive)
				{
					Errors(&ErrorMgr, ERROR_PENDANT, ERROR_ADROID_COM_LOST, 0);
					LogTxt(&LogMgr, "Pendant com. error");
					TML_MTR_CUT_POWER = 1;

					KK_CatchAndroidComErr = AndroidConnect_Tmr.ET;
					KK_CatchAndroidErr	= 1;
				}

				m->AndIntrf[0].Alive = 0;

			}

		}
		else
		{

			AndroidConnect_Tmr.IN = 0;
			AndroidConnect_Tmr.Q = 0;

		}

	}

	///////////////////////////////////////////////
	//	ESTOP and ERROS handling

	if (m->pESTOP_Inp)
	{

#ifdef TEST_ONLY_PLC_ANDROID
		(*m->pESTOP_Inp)	= 1;					// Remove KK
#endif
		if(!(*m->pESTOP_Inp))
		{
			//ESTOP_Inp_Status = 1;
			m->ESTOP			= 1;
			ESTOP_Dly_Tmr.IN	= 0;
			ESTOP_Dly_Tmr.Q		= 0;
			Ready2StoreLastPos = 0;

			if ((m->sm.Step > 5 && m->sm.Step < 190) || (m->sm.Step == 0) || (m->sm.Step == 1))
			{
				Errors(&ErrorMgr,ERROR_ESTOP,ERROR_ESTOP_ERR,1);
				TML_MTR_CUT_POWER = 1;
				m->sm.Step	= 190;
			}

			// This is only when you have to clear Estop then clear error - not opposite
			if(!ErrorMgr.Error)
				Errors(&ErrorMgr,ERROR_ESTOP,ERROR_ESTOP_ERR,1);

		}
		else {

			ESTOP_Inp_Status = 0;

			if(ProjectConfig == project_US_Orbital)
				m->ESTOP = TML_MTR_CUT_POWER;

			else{

				//ESTOP_Dly_Tmr.IN	= !TML_MTR_CUT_POWER;
				//m->ESTOP = !ESTOP_Dly_Tmr.Q;

				m->ESTOP = 0;

			}
		}

	}

	if (ErrorMgr.Error && !m->LOCKED && !KK_ErrorsHold)
	{

		if (m->sm.Step > 5 && m->sm.Step < 190)
		{ // Give chance to clear error by step first steps and download TML programs

			// Always Coolant On
			if (Process[m->pCfg->HeadCfg.COOL.PROC_Indx].Status != prcsSTATUS_Run)
				Process[m->pCfg->HeadCfg.COOL.PROC_Indx].xCMD = prcsSTART;

			Process[m->pCfg->HeadCfg.TVL.PROC_Indx].xCMD = prcsHalt;
			Process[m->pCfg->HeadCfg.OSC.PROC_Indx].xCMD = prcsHalt;
			Process[m->pCfg->HeadCfg.AVC.PROC_Indx].xCMD = prcsHalt;
			Process[m->pCfg->HeadCfg.WF.PROC_Indx].xCMD = prcsHalt;
			Process[m->pCfg->HeadCfg.WP.PROC_Indx].xCMD = prcsHalt;
			Process[m->pCfg->HeadCfg.TIG.PROC_Indx].xCMD = prcsHalt;
			Process[m->pCfg->HeadCfg.HW.PROC_Indx].xCMD = prcsHalt;

			Process[m->pCfg->HeadCfg.GAS.PROC_Indx].xCMD = prcsSTOP;

			//Process[m->pCfg->HeadCfg.COOL.PROC_Indx].xCMD = prcsHalt;
			m->Mode 			= MASTER_MODE_ERROR;

			Ready2StoreLastPos = 0;
			m->sm.Step			= 200;

		}

	}

	////////////////////////////////////////////////////////////////
	// Extra Imperatives
	//curCfg->Param[parTVL_RunDist].val[0] = (float)curCalib->GenSetup[SETUP_TVL_DISTANCE];
	///////////////////////////////////////////////////////////////
	KK_HomeBtn			= (!intrf->_intr._GlblBtnCmd[0] && (intrf->GlblBtnCmd[0] &ANDR_BTN_HOME));
	KK_StopBtn			= (!intrf->_intr._GlblBtnCmd[0] && (intrf->GlblBtnCmd[0] &ANDR_BTN_STOP));

	if((intrf->GlblBtnCmd[0] & ANDR_BTN_HOME) && (intrf->GlblBtnCmd[0] &ANDR_BTN_STOP))
		Weld_Report_Status = 0;

	// MAIN STATES //
	switch (m->sm.Step)
	{
		case 0:	sm_text("Start", &m->sm);

			Ready2StoreLastPos = 0;

		#ifndef MIG_PENDANT

			if (ANDROID_Pendant)
			{ // start only when is android connection

				if (_datagramCountTotal[0] == datagramCountTotal[0]){
					//TML_MTR_CUT_POWER = 1;
					break;
				}

			}

		#endif

			if(intrf->GlblBtnCmd[0] & (0xFFFFFFFF
					-ANDR_BTN_STOP -0x04000000 - 0x10000000 - 0x20000000 - 0x02000000 - 0x08000000 )){

				strcpy(hmi->pMessage[0], " DO NOT HOLD BUTTON");
				strcpy(hmi->pMessage[1], " ");
				strcpy(hmi->pMessage[2], " ");
				strcpy(hmi->pMessage[3], " ");
				TimerStart(&hmi->MsgTmr, 1.0);

				break;

			}
			else if (ErrorMgr.Error && !KK_Functionality && !KK_ErrorsHold)
			{

				m->Mode 			= MASTER_MODE_ERROR;
				break;
			}

			else if (!intrf->_intr._GlblBtnCmd[0] && (intrf->GlblBtnCmd[0] & ANDR_BTN_STOP))
			{
				//AckAllErrors(&ErrorMgr);

			}

			else if (m->ESTOP)
			{

				m->Mode 			= MASTER_MODE_ESTOP;

				break;
			}

			hmi->Node2JumpID = P_MODE_1;
			//hmi->JumpLineID = 0;
			//hmi->xCMD = JUMP2ID_CMD;
			hmi->DynPageNodeIndx = 0xFFFF;
			lcd->StaticMessageVisible = 0;
			ParametrAssignToPointers(m, m->curSegm[ZONE]);
			intrf->ModeLED = 1;
			PleaseUpdateHeadSetup(m);
			//AckAllErrors(&ErrorMgr);
			TML_MTR_CUT_POWER = 0;

			/*
			for (i = 0; i < PROCESS_NUM; i++)
				Process[i].xCMD = prcsRESTART;

			for (i = 0; i < TML_SERVO_NUM; i++)
			{

				TML_MTR_INST[i].xCMD = TML_RESTART;
				TML_MTR_INST[i]._int.restartCnt = 0;
				TML_MTR_INST[i]._int.Init = 0;
			}
			*/

			TML_Restart_Step = 1;
			Process_Restart_Step = 0;

			m->SeqStep = 0;
			m->Mode = MASTER_MODE_INIT;

			if(curCalib->GenSetup[SETUP_INDX_ENBL] == 0
				|| curCalib->GenSetup[SETUP_INDX_ENBL] == 3){ // Not Installed or OSC Index

				if( m->pCfg->HeadCfg.INDX.VECT_A_Indx > 0)
					VectorStateMach[m->pCfg->HeadCfg.INDX.VECT_A_Indx].simul = 1;

				if( m->pCfg->HeadCfg.INDX.VECT_B_Indx > 0)
					VectorStateMach[m->pCfg->HeadCfg.INDX.VECT_B_Indx].simul = 1;

				if(m->pCfg->HeadCfg.INDX.TML_A_Indx > 0)
					TML_MTR_INST[m->pCfg->HeadCfg.INDX.TML_A_Indx].Disable = 1;

				if(m->pCfg->HeadCfg.INDX.TML_B_Indx > 0)
					TML_MTR_INST[m->pCfg->HeadCfg.INDX.TML_B_Indx].Disable = 1;

			}else{

				if( m->pCfg->HeadCfg.INDX.VECT_A_Indx > 0)
					VectorStateMach[m->pCfg->HeadCfg.INDX.VECT_A_Indx].simul = 0;

				if( m->pCfg->HeadCfg.INDX.VECT_B_Indx > 0)
					VectorStateMach[m->pCfg->HeadCfg.INDX.VECT_B_Indx].simul = 0;

				if(m->pCfg->HeadCfg.INDX.TML_A_Indx > 0)
					TML_MTR_INST[m->pCfg->HeadCfg.INDX.TML_A_Indx].Disable = 0;

				if(m->pCfg->HeadCfg.INDX.TML_B_Indx > 0)
					TML_MTR_INST[m->pCfg->HeadCfg.INDX.TML_B_Indx].Disable = 0;

			}

			// Coolant always ON
			//Process[m->pCfg->HeadCfg.COOL.PROC_Indx].xCMD = prcsForceON;
			curTML_indx = 0;
			//TimerStart(&m->sm.Tmr1, 4.0); // Time to Init TML servo
			TimerStart(&m->sm.Tmr1, 4.0); // Time to Init TML servo
			//Hold_Estop_ON = 0;
			m->LOCKED = 0;
			m->sm.Step++;

		break;

		case 1:	sm_text("Check TML", &m->sm);

			//TML_STOP_SEND_ERROR = 0;

			if(!((TML_Restart_Step == 0) && (Process_Restart_Step == 0)))
				break;

			if (TimerIsTimeOut(&m->sm.Tmr1))
			{ // Check why TML did not start

				status				= 0;
				_status 			= status;

				for (i = 0; i < TML_SERVO_NUM; i++)
				{

					if (TML_MTR_INST[i].pState && !TML_MTR_INST[i].Disable)
					{

						if (TML_MTR_INST[i].xCMD == TML_WAIT_FOR_DOWNLOAD)
						{

							LogTxt(&LogMgr, "Wrong Setup %s ", TML_MTR_INST[i].Name);

							if (_status < 2)
								status = 2;

						}

						else if (TML_MTR_INST[i]._int.restartCnt > 10)
						{

							LogTxt(&LogMgr, "CAN com. Err. %s ", TML_MTR_INST[i].Name);
							if(TML_MTR_INST[i].ErrorReg)
								Errors(&ErrorMgr ,ERROR_MOTOR , ERROR_DRV_01 + i , 17);
							else
								Errors(&ErrorMgr ,ERROR_MOTOR , ERROR_DRV_01 + i , 18);

							if (_status < 1)
								status = 1;

						}
						else if (!TML_MTR_INST[i]._int.Init)
						{

#ifndef TEST_ONLY_PLC_ANDROID

							if (TML_MTR_INST[i].xCMD)
								LogTxt(&LogMgr, "Not Comun. %s ", TML_MTR_INST[i].Name);
							else
								LogTxt(&LogMgr, "Not Init. %s ", TML_MTR_INST[i].Name);

							if(TML_MTR_INST[i].ErrorReg)
								//Errors(&ErrorMgr ,ERROR_MOTOR , ERROR_TML_1 + i , TML_MTR_INST[i].ErrorReg);
								Errors(&ErrorMgr ,ERROR_MOTOR , ERROR_DRV_01 + i , 17);
							else
								Errors(&ErrorMgr ,ERROR_MOTOR , ERROR_DRV_01 + i , 18);

							if (_status < 1)
								status = 1;

#endif
						}

						_status 			= status;

					}

				}

			}
			else
			{

				status				= 1;

				for (i = 0; i < TML_SERVO_NUM; i++)
				{

					if (TML_MTR_INST[i].pState)
					{

						if (!TML_MTR_INST[i]._int.Init)
							status = 0;

					}

				}

				if (status)
				{
					m->sm.Step			= 5;
					break;
				}
				else
					break;

			}

			if (KK_DoNotChangeTMLProgram)
			{
				if (status == 2)
					status = 0;
			}

			KK_actPosProcss = status;

			switch (status)
			{
				case 1:

					//Errors(&ErrorMgr, ERROR_MOTOR, ERROR_TML_1, 10);

					// Display which one has error in previous step

					if(!KK_ErrorsHold){

						TML_MTR_CUT_POWER = 1;
						m->sm.Step = 200;
					}
					else{

						if (ANDROID_Pendant){

							m->sm.Step = 5;

						}
						else
						{

							TimerStart(&m->sm.Tmr1, 5.0); // Time to Init Arclink
							m->sm.Step	= 49;

						}

					}

				break;

				case 2:

					if(!KK_ErrorsHold){

						TML_MTR_CUT_POWER = 1;
						m->LOCKED = 1;
					}
					else{

						if (ANDROID_Pendant){

							m->sm.Step = 5;

						}
						else
						{

							TimerStart(&m->sm.Tmr1, 5.0); // Time to Init Arclink
							m->sm.Step	= 49;

						}
					}

				break;

				default:

					if (ANDROID_Pendant){

						m->sm.Step = 5;

					}
					else
					{

						TimerStart(&m->sm.Tmr1, 5.0); // Time to Init Arclink
						m->sm.Step	= 49;

					}

				break;
			}

			break;

		case 5:	sm_text("W: Pendant ", &m->sm);

			 TML_STOP_SEND_ERROR = 0;

			//if(datagramCountTotal[0] > 100)
//#ifndef TEST_ONLY_PLC_ANDROID

			//if (m->AndIntrf[0].Alive)
//#else

				//if(1)
//#endif

				if(1){

					KK_AUTO_Test		= 0;

					TimerStart(&DoubleStop_TMR, 0.1);
					ParametrAssignToPointers(m, m->curSegm[ZONE]);

					m->SubSeqStep = 1;

					TimerStart(&m->sm.Tmr1, 60.0);		// Time to Init Arclink
					m->sm.Step			= 49;

				}

				////////////////////////////////////

				if(KK_FirstRestart_Loop){

					KK_FirstRestart_Loop --;
					m->sm.Step = 0;

				}
		break;

		case 49: sm_text("W: Arclink PS Rdy", &m->sm);

			//Hold_Estop_ON = 0;

			//if(strlen(ArcLinkPS_IP_Address) == 0){
			if(PS_Param_Set[0].Mode == 0){ // NO Arclink

				SetTVL_Pos_Feedback();

				MV[0].xCMD = MV_RESTART_CMD;

				for (i = 0; i < PROCESS_NUM; i++)
					Process[i].fParam[0] = 0.0;

				if(!intrf->GlblBtnCmd[0])
					m->sm.Step = 50;

				break;

			}
			else if (robot)
			{ // Arclink connection

				if (robot->Cntrl.Fbk.Status & PS_Ready){
					SetTVL_Pos_Feedback();
					TVL_Latch_Latched = 0;

					MV[0].xCMD = MV_RESTART_CMD;

					for (i = 0; i < PROCESS_NUM; i++)
						Process[i].fParam[0] = 0.0;

					if(!intrf->GlblBtnCmd[0])
						m->sm.Step = 50;

				}
				else if(TimerIsTimeOut(&m->sm.Tmr1)){

					Errors(&ErrorMgr,ERROR_TIG_PROC, ERROR_ARCLINK_COM_LOST, 1 );
					LogTxt(&LogMgr , "Arclink TimeOut "  );

				}

			}
			else {
				SetTVL_Pos_Feedback();
				TVL_Latch_Latched = 0;

				MV[0].xCMD = MV_RESTART_CMD;

				for (i = 0; i < PROCESS_NUM; i++)
					Process[i].fParam[0] = 0.0;

				if(!intrf->GlblBtnCmd[0])
					m->sm.Step = 50;
			}

		break;

		// Watch for button pressed
		case 50: sm_text("Normal Stop", &m->sm);

			Ready2StoreLastPos = 1;

			if(PS_Param_Set[0].Mode){
				if (WatchArcLinkError(m, robot))
					break;
			}

			m->Mode = MASTER_MODE_STOP;

			if (_curZone != m->curSegm[ZONE])
				ParametrAssignToPointers(m, m->curSegm[ZONE]);

			_curZone = m->curSegm[ZONE];

			StopModeAndroidButtons(m, hmi, &HMI_Intr, lcd);
			StopModeAndroidButtons(m, hmi, intrf, lcd);

			StartBtn = (!intrf->_intr._GlblBtnCmd[0] && (intrf->GlblBtnCmd[0] &ANDR_BTN_START));
			StopBtn = (!intrf->_intr._GlblBtnCmd[0] && (intrf->GlblBtnCmd[0] &ANDR_BTN_STOP));
			/// was added on March 28 , 2019///
			if(StopBtn){
				TVL_Latch_Latched = 0;
				_TVL_Latch_Latched	= TVL_Latch_Latched;

			}
			///////
			TVL_ROT_Param_Set[0].HeadSwitch = (curCfg->Param_ENUM[parENUM_PathMode].val[0] == 0.0)? 1:0;
			TVL_ROT_Param_Set[0].Extras = (UINT)(curCalib->GenSetup[SETUP_EXTRAS]);

			switch(curCalib->GenSetup[SETUP_CONTIN_WELD]){

				case 1: // CONTINUE ONE WAY

					MasterSequence_Contin_OneWay(m, hmi, StartBtn, StopBtn);

				break;

				case 2: // CONTINUE BOTH DIRECTION

					MasterSequence_Contin(m, hmi, StartBtn, StopBtn);

				break;

				default: // STANDARD

					MasterSequence(m, hmi, StartBtn, StopBtn);

				break;

			}

			hmi->CalibMode = 0; // No Calibration

			if(m->SeqStep > 0)
				m->sm.Step = 51;

		break;

		case 51:
			sm_text("Normal Run", &m->sm);

			if(PS_Param_Set[0].Mode){
				if (WatchArcLinkError(m, robot))
					break;
			}

			m->Mode = MASTER_MODE_RUN;

			if (_curZone != m->curSegm[ZONE])
				ParametrAssignToPointers(m, m->curSegm[ZONE]);

			_curZone = m->curSegm[ZONE];

			//if (Process[m->pCfg->HeadCfg.AVC.PROC_Indx].Status != prcsSTATUS_Stopped )
			if ((Process[m->pCfg->HeadCfg.AVC.PROC_Indx].Status != prcsSTATUS_Stopped)
				|| (m->TestMode))
				RunModeAndroidButtons(m, hmi, intrf, lcd);
			else
				StopModeAndroidButtons(m, hmi, intrf, lcd);

			StartBtn = (!intrf->_intr._GlblBtnCmd[0] && (intrf->GlblBtnCmd[0] &ANDR_BTN_START));
			StopBtn = (!intrf->_intr._GlblBtnCmd[0] && (intrf->GlblBtnCmd[0] &ANDR_BTN_STOP));

			//MasterSequence(m, hmi, StartBtn, StopBtn);

			switch(curCalib->GenSetup[SETUP_CONTIN_WELD]){

				case 1: // CONTINUE ONE WAY

					MasterSequence_Contin_OneWay(m, hmi, StartBtn, StopBtn);

				break;

				case 2: // CONTINUE BOTH DIRECTION

					Weld_Report_Status = 2; // Always ready to acknowledge
					MasterSequence_Contin(m, hmi, StartBtn, StopBtn);

				break;

				default: // STANDARD

					MasterSequence(m, hmi, StartBtn, StopBtn);

				break;

			}

			if (m->SeqStep == 0)
				m->sm.Step = 50;

		break;

		case 100:	sm_text("Calibration Stop", &m->sm);

			Ready2StoreLastPos = 1;

			m->Mode = MASTER_MODE_CALIB_STOP;
			StopCalibrationModeAndroidButtons(m, hmi, intrf, lcd);
			StartBtn = (!intrf->_intr._GlblBtnCmd[0] && (intrf->GlblBtnCmd[0] &ANDR_BTN_START));
			StopBtn = (!intrf->_intr._GlblBtnCmd[0] && (intrf->GlblBtnCmd[0] &ANDR_BTN_STOP));

			switch (CalibrationSequence(m, hmi, StartBtn, StopBtn))
			{
				case 0: // Not Ready
				break;

				case 1: //	Stop

				break;

				case 2: //	Run
					m->sm.Step = 101;
				break;
			}

		break;

		case 101: sm_text("Calibration Run", &m->sm);

			m->Mode = MASTER_MODE_CALIB_RUN;
			RunCalibrationModeAndroidButtons(m, hmi, intrf, lcd);
			StartBtn = (!intrf->_intr._GlblBtnCmd[0] && (intrf->GlblBtnCmd[0] &ANDR_BTN_START));
			StopBtn = (!intrf->_intr._GlblBtnCmd[0] && (intrf->GlblBtnCmd[0] &ANDR_BTN_STOP));

			switch (CalibrationSequence(m, hmi, StartBtn, StopBtn))
			{
				case 0: // Not Ready
					m->sm.Step = 100;
				break;

				case 1: //	Stop
					m->sm.Step = 100;
				break;

				case 2: //	Run

					DrillDwnHMI.StartBtn_Vis = 0 ; //VISIBLE;
					DrillDwnHMI.StopBtn_Vis = 0 ; //VISIBLE;

				break;
			}

		break;

		////////////////////////////////////////
		////////////////////////////////////////
		case 190: sm_text("ESTOP Catched!", &m->sm);

			m->Mode = MASTER_MODE_ESTOP;

			TVL_Latch_Latched = 0;

			LogMgr.Cmd.PauseLog = 0;

			/*
			hmi->Node2JumpID = P_INIT;
			hmi->JumpLineID = 0;
			hmi->xCMD = JUMP2ID_CMD;
			hmi->DynPageNodeIndx = P_INIT;
			*/
			LogTxt(&LogMgr, " ESTOP Pressed");

			for (i = 0; i < PROCESS_NUM; i++){

				if(i == m->pCfg->HeadCfg.GAS.PROC_Indx)
					Process[i].xCMD = prcsSTOP;
				else
					Process[i].xCMD = prcsHalt;

			}

			Process[m->pCfg->HeadCfg.COOL.PROC_Indx].xCMD = prcsSTOP;
			Process[m->pCfg->HeadCfg.GAS.PROC_Indx].xCMD = prcsSTOP; // remain gas
			m->SeqStep = 0;
			ParametrAssignToPointers(m, m->curSegm[ZONE]);

			TimerStart(&m->sm.Tmr1, 2.5);

			m->sm.Step++;

		break;

		case 191: sm_text("Wait: ESTOP", &m->sm);

			if(!TimerIsTimeOut(&m->sm.Tmr1))
				break;

			TML_MTR_CUT_POWER = 0; // To Wazne i grozne

			if (!m->ESTOP)
			{

				TVL_Latch_Latched = 0;

				if(!intrf->GlblBtnCmd[0]){

					if(ErrorMgr.Error){

						if(KK_Functionality)
							m->sm.Step = 0;
						else
							m->sm.Step = 200;

					}
					else{

#ifdef TML_CMD_LOGS

						memset(&Cmd_Log_Mgr , 0 , sizeof(Cmd_Log_Mgr));
						Cmd_Log_Mgr.AxisID_filter = AxisID_filter;
#endif

						m->sm.Step = 0;

					}

				}else {

					strcpy(hmi->pMessage[0], " DO NOT HOLD BUTTON");
					strcpy(hmi->pMessage[1], " ");
					strcpy(hmi->pMessage[2], "It is recovery");
					strcpy(hmi->pMessage[3], "after ESTOP");
					TimerStart(&hmi->MsgTmr, 1.0);

				}

			}
			else if(m->pESTOP_Out){ // For US Orbital only - allow to clear ESTOP
				TML_MTR_CUT_POWER = 0;
				TML_STOP_SEND_ERROR = 1;

			}
			else
				TML_STOP_SEND_ERROR = 1;

		break;

		////////////////////////////////////////
		////////////////////////////////////////
		case 200: sm_text("ERROR !", &m->sm);

			m->Mode = MASTER_MODE_ERROR;

			if (m->sm.Step != m->sm.oldStep)
			{

				if (!m->ESTOP)
					hmi->DynPageNodeIndx = P_ERRORS;

				LogTxt(&LogMgr, " Get ERROR ");

			}
			else if (ErrorMgr.Error <= ERROR_FATAL)
			{
				hmi->DynPageNodeIndx = P_ERRORS;
				m->sm.Step			= 255;

			}
			else if (!ErrorMgr.Error)
			{
				m->Mode 			= MASTER_MODE_INIT;

				if(!(intrf->GlblBtnCmd[0] & (0xFFFFFFFF -ANDR_BTN_STOP))){

					//////////////////////////
					if (robot)
					{ // Arclink connection

						if (robot->Cntrl.Fbk.Error > 0)
							robot->Cntrl.Cmd.RST = 1;

					}
					/////////////////////////
					TimerStart(&m->sm.Tmr1, 3.0);

					TML_MTR_CUT_POWER = 0;

					TVL_Latch_Latched = 0;

					//for (i = 0; i < TML_SERVO_NUM; i++)
						//TML_MTR_INST[i].xCMD = TML_RESTART;

					m->sm.Step++;

				}

			}
			/*
			else if(intrf->GlblBtnCmd[0] & (0xFFFFFFFF - ANDR_BTN_ENTER
					-ANDR_BTN_STOP -0x04000000 - 0x10000000 - 0x20000000 - 0x02000000 - 0x08000000   )){ // all butons excludes navigation buttons

					strcpy(hmi->pMessage[0], " DO NOT HOLD BUTTON");
					strcpy(hmi->pMessage[1], "");
					strcpy(hmi->pMessage[2], "It is ERROR state");
					strcpy(hmi->pMessage[3], "");
					TimerStart(&hmi->MsgTmr, 1.0);

			}
			*/
			else if (!intrf->_intr._GlblBtnCmd[0] && (intrf->GlblBtnCmd[0] & ANDR_BTN_STOP))
			{

					KK_test++;
					AckAllErrors(&ErrorMgr);

			}

			if(m->ESTOP)
				m->sm.Step = 190;

		break;

		case 201: sm_text("No Errors wait", &m->sm);

#ifdef MIG_EXP_SYSTEM

			if(Kick_TML_Cmd != 0)
				break;

#endif

			if (TimerIsTimeOut(&m->sm.Tmr1))
			{
				/*
				hmi->Node2JumpID	= P_MODE_1;
				hmi->JumpLineID 	= 0;
				hmi->xCMD			= JUMP2ID_CMD;
				*/

				/*
				TVL_Latch_Latched = 0;

				for (i = 0; i < TML_SERVO_NUM; i++)
					TML_MTR_INST[i].xCMD = TML_RESTART;
				*/

				m->sm.Step			= 0;

				#ifdef NG4_TIG_SYSTEM
				KK_FirstRestart_Loop = 1;
				#else
				KK_FirstRestart_Loop = 0;
				#endif

			}

		break;

		////////////////////////////////////////////
		/////  New Head Configuration Selected
		case 230: sm_text("Please Clear Estop", &m->sm);

			/*
			Hold_Estop_ON = 1;
			TML_MTR_CUT_POWER = 0;

			if (!ESTOP_Inp_Status)
				m->sm.Step++;
			*/

			//TML_MTR_CUT_POWER = 1;
			//TML_STOP_SEND_ERROR = 1;
			//m->LOCKED = 1;

			m->LOCKED = 1;
			TML_MTR_CUT_POWER = 1;
			TML_STOP_SEND_ERROR = 1;

			if(m->ESTOP
				|| (ProjectConfig == project_FourAxisTig)){

				LogTxt(&LogMgr, "Checking TML Setup");

				m->sm.Step++;

			}

		break;

		case 231: sm_text("Check (2) TML", &m->sm);

			if(!intrf->_intr._GlblBtnCmd[0] && (intrf->GlblBtnCmd[0] &ANDR_BTN_START)){

				for (i = 0; i < TML_SERVO_NUM; i++){

					TML_MTR_INST[i]._int.restartCnt = 0;
					TML_MTR_INST[i]._int.Init = 0;
					TML_MTR_INST[i].xCMD = TML_RESTART;

				}

				TimerStart(&m->sm.Tmr1, 4.0);

				m->sm.Step++;

			}

			else if(!intrf->_intr._GlblBtnCmd[0] && (intrf->GlblBtnCmd[0] &ANDR_BTN_STOP)){

				m->sm.Step = 999;

			}

		break;

		case 232: sm_text("Check TML (3)", &m->sm);

			if(ESTOP_Inp_Status){
				m->sm.Step = 230;
				break;
			}

			if (TimerIsTimeOut(&m->sm.Tmr1))
			{

				status	= 0;

				for (i = 0; i < TML_SERVO_NUM; i++)
				{

					if (TML_MTR_INST[i].pState && !TML_MTR_INST[i].Disable)
					{

						if (status == 0)
						{ // Catch only first

							if(TML_MTR_INST[i].xCMD)
							{
								/*
								if (((TML_MTR_INST[i].xCMD == TML_WAIT_FOR_DOWNLOAD) || (TML_MTR_INST[i].xCMD <= 9))
									&& (!TML_MTR_INST[i]._cfg.NotAutoDownload))
								{ // Reset was blocked
									curTML_indx = i;
									status = 1;
								}
								*/

								if ((TML_MTR_INST[i].xCMD == TML_WAIT_FOR_DOWNLOAD) || (TML_MTR_INST[i].xCMD <= 9))

								{
									curTML_indx = i;
									if((!TML_MTR_INST[i]._cfg.NotAutoDownload) || KK_Can_Download_Everything ){
										//curTML_indx = i;
										status = 1;
									}
									else{

										LogTxt(&LogMgr, "Change %s Setup only in Diagn. ", TML_MTR_INST[curTML_indx].Name);

										strcpy(hmi->pMessage[0], "Setup Change of");
										strcpy(hmi->pMessage[1], TML_MTR_INST[curTML_indx].Name);
										xsprintf(hmi->pMessage[2], "can be done");
										strcpy(hmi->pMessage[3], "only in Diagnostic");
										TimerStart(&hmi->MsgTmr, 3.0);

										status = 2;

									}

								}
							}

						}
					}

				}

				if (status == 1)
					m->sm.Step++;
					//m->sm.Step = 1999;

				else if (status == 2)
					m->sm.Step = 230;
					//m->sm.Step = 1999;

				else
				{
					m->sm.Step = 246;
				}

			}

		break;

		case 233: sm_text("Start Download", &m->sm);

			if(ESTOP_Inp_Status){
				m->sm.Step = 230;
				break;
			}

			m->LOCKED = 1;
			TML_MTR_CUT_POWER = 1;
			TML_STOP_SEND_ERROR = 1;

			if(m->ESTOP
				|| (ProjectConfig == project_FourAxisTig)){

				if(!intrf->_intr._GlblBtnCmd[0] && (intrf->GlblBtnCmd[0] &ANDR_BTN_START)){

					/*
					m->LOCKED = 1;
					TML_MTR_CUT_POWER = 1;
					TML_STOP_SEND_ERROR = 1;
					*/

					if(TML_Setup_From_Diagn)
						m->LOCKED = 1;

					if (File_RW.CMD == 0)
					{
						TML_MTR_INST[curTML_indx].xCMD = TML_DOWNL;
						TimerStart(&m->sm.Tmr1, 30.0);
						m->sm.Step++;
					}
					else
					{
						LogTxt(&LogMgr, "File Manager busy");
						m->sm.Step			= 1;
					}

				}
				else if(!intrf->_intr._GlblBtnCmd[0] && (intrf->GlblBtnCmd[0] &ANDR_BTN_STOP)){

					m->sm.Step = 999;

				}
			}

		break;

		case 234: sm_text("Wait Downloading", &m->sm);

			if(ESTOP_Inp_Status){
				m->sm.Step = 230;
				break;
			}

			if (TML_MTR_INST[curTML_indx].xCMD == 107)
			{
				TimerStart(&m->sm.Tmr1, 4.0);
				m->sm.Step = 235;
			}
			else if (TML_MTR_INST[curTML_indx].xCMD == 106)
			{
				TimerStart(&m->sm.Tmr1, 4.0);
				m->sm.Step = 236;
			}
			else if ((TML_MTR_INST[curTML_indx].xCMD == TML_DOWNL_DONE)
				|| (TML_MTR_INST[curTML_indx].xCMD == TML_IDLE)){

				LogTxt(&LogMgr, "%s Setup is Uploaded" ,TML_MTR_INST[curTML_indx].Name );
				m->sm.Step = 245;

			}

			else if (TimerIsTimeOut(&m->sm.Tmr1)){

				LogTxt(&LogMgr, "%s Load Setup TimeOut" ,TML_MTR_INST[curTML_indx].Name );

				strcpy(hmi->pMessage[0], "Setup Download To");
				strcpy(hmi->pMessage[1], TML_MTR_INST[curTML_indx].Name);
				xsprintf(hmi->pMessage[2], "is Timeouted");
				strcpy(hmi->pMessage[3], " ");
				TimerStart(&hmi->MsgTmr, 3.0);

				m->sm.Step = 246;

			}

		break;

		case 235:  sm_text("Wait Downloading1", &m->sm);

			if(ESTOP_Inp_Status){
				m->sm.Step = 230;
				break;
			}

			if (TML_MTR_INST[curTML_indx].xCMD != 107)
			{
				m->sm.Step = 234;
			}
			else if (TimerIsTimeOut(&m->sm.Tmr1))
			{
				//TML_MTR_INST[curTML_indx].xCMD = TML_DOWNL;
				LogTxt(&LogMgr, "Setup Transm. Error %s", TML_MTR_INST[curTML_indx].Name);
				m->sm.Step = 230;
			}

		break;

		case 236:

			if(ESTOP_Inp_Status){
				m->sm.Step = 230;
				break;
			}

			if (TML_MTR_INST[curTML_indx].xCMD != 106)
			{
				m->sm.Step = 234;
			}
			else if (TimerIsTimeOut(&m->sm.Tmr1))
			{
				LogTxt(&LogMgr, "Setup Transm. Error %s", TML_MTR_INST[curTML_indx].Name);
				m->sm.Step = 230;
			}

		break;

		case 245: // Try again setup checkout

			if(TML_Setup_From_Diagn){
				TML_Setup_From_Diagn = 0;
				m->sm.Step = 222; // Got o to step 0
				//m->sm.Step = 1000; // Freeze and wait for Restart
			}
			else
				m->sm.Step = 231;
		break;

		case 246: // Restart Whole system <Manually

			/*
			if(TML_Setup_From_Diagn){
				m->sm.Step = 1000; // Freeze and wait for Restart
			}
			else
				m->sm.Step = 999; // Freeze and wait for Restart
			*/

			TML_Setup_From_Diagn = 0;
			//m->sm.Step = 222; // Got o to step 0
			m->LOCKED = 0;
			m->sm.Step = 0;
			//m->xCmd = 1; //Restart entire system

			TML_Setup_From_Diagn = 0;
		break;

		case 250: // SYSTEM MUST BE RESTARTED = Power Cyclic

			sm_text("Head Restarted 0", &m->sm);

			LogTxt(&LogMgr, "Heasd Setup Change - must reboot");

			strcpy(hmi->pMessage[0], "Head Setup");
			strcpy(hmi->pMessage[1], "Changed");
			xsprintf(hmi->pMessage[2], "Please");
			strcpy(hmi->pMessage[3], "Power OFF/ON");
			TimerStart(&hmi->MsgTmr, 3.0);

			TML_MTR_CUT_POWER = 1;

			m->sm.Step++;

		break;

		case 251:

			sm_text("Head Restarted 1", &m->sm);

			SYSTEM_LOCKED = 1;

		break;

		case 999:  sm_text("Dead End 999", &m->sm);

		break;

		case 1000:  sm_text("Dead End 1000", &m->sm);

		break;

		case 1001:  sm_text("Dead End 1001", &m->sm);

		break;

	}

		// Head Selection
		// FWD Direction  - Head B	m->ToolHeadID = 1
		if (m->ToolHeadID == 0)
		{
			Hardware[1].Outp[5] = 1;	// Select A Head Signal
			Hardware[1].Outp[0] = 1;	// Weld Angle

			//TVL
			Process[m->pCfg->HeadCfg.TVL.PROC_Indx].Param[1] = 0; // Select Calibration & Direction

			if(curCalib->GenSetup[SETUP_WF_WP_SWAP] == 0){

				//WF
				Process[m->pCfg->HeadCfg.WF.PROC_Indx].Param[1] = 0; // Select Calibration

				if(m->pCfg->HeadCfg.WF.VECT_A_Indx > 0)
					WIRE_Param_Set[0].pVect = &VectorStateMach[m->pCfg->HeadCfg.WF.VECT_A_Indx];
				else
					WIRE_Param_Set[0].pVect = 0;

				if(m->pCfg->HeadCfg.WF.VECT_A_Indx != m->pCfg->HeadCfg.WF.VECT_B_Indx){

					if(m->pCfg->HeadCfg.WF.VECT_B_Indx > 0)
						VectorStateMach[m->pCfg->HeadCfg.WF.VECT_B_Indx].InVal = 0.0;
				}

				if(m->pCfg->HeadCfg.WF.VECT_Aux_A_Indx > 0)
					WIRE_Param_Set[0].pAuxVect = &VectorStateMach[m->pCfg->HeadCfg.WF.VECT_Aux_A_Indx];
				else
					WIRE_Param_Set[0].pAuxVect = 0;

				if(m->pCfg->HeadCfg.WF.VECT_Aux_A_Indx != m->pCfg->HeadCfg.WF.VECT_Aux_B_Indx){

					if(m->pCfg->HeadCfg.WF.VECT_Aux_B_Indx > 0)
						VectorStateMach[m->pCfg->HeadCfg.WF.VECT_Aux_B_Indx].InVal = 0.0;
				}

				//WP
				Process[m->pCfg->HeadCfg.WP.PROC_Indx].Param[1] = 0; // Select Calibration

				if(m->pCfg->HeadCfg.WP.VECT_A_Indx > 0)
					WIRE_Param_Set[1].pVect = &VectorStateMach[m->pCfg->HeadCfg.WP.VECT_A_Indx];
				else
					WIRE_Param_Set[1].pVect = 0;

				if(m->pCfg->HeadCfg.WP.VECT_A_Indx != m->pCfg->HeadCfg.WP.VECT_B_Indx){

					if(m->pCfg->HeadCfg.WP.VECT_B_Indx > 0)
						VectorStateMach[m->pCfg->HeadCfg.WP.VECT_B_Indx].InVal = 0.0;
				}

			}
			else{

				//WF
				Process[m->pCfg->HeadCfg.WF.PROC_Indx].Param[1] = 1; // Select Calibration

				if(m->pCfg->HeadCfg.WF.VECT_B_Indx > 0)
					WIRE_Param_Set[0].pVect = &VectorStateMach[m->pCfg->HeadCfg.WF.VECT_B_Indx];
				else
					WIRE_Param_Set[0].pVect = 0;

				if(m->pCfg->HeadCfg.WF.VECT_A_Indx != m->pCfg->HeadCfg.WF.VECT_B_Indx){

					if(m->pCfg->HeadCfg.WF.VECT_A_Indx > 0 )
						VectorStateMach[m->pCfg->HeadCfg.WF.VECT_A_Indx].InVal = 0.0;
				}

				if(m->pCfg->HeadCfg.WF.VECT_Aux_B_Indx > 0)
					WIRE_Param_Set[0].pAuxVect = &VectorStateMach[m->pCfg->HeadCfg.WF.VECT_Aux_B_Indx];
				else
					WIRE_Param_Set[0].pAuxVect = 0;

				if(m->pCfg->HeadCfg.WF.VECT_Aux_A_Indx != m->pCfg->HeadCfg.WF.VECT_Aux_B_Indx){

					if(m->pCfg->HeadCfg.WF.VECT_Aux_A_Indx > 0)
						VectorStateMach[m->pCfg->HeadCfg.WF.VECT_Aux_A_Indx].InVal = 0.0;
				}

				//WP
				Process[m->pCfg->HeadCfg.WP.PROC_Indx].Param[1] = 1; // Select Calibration

				if(m->pCfg->HeadCfg.WP.VECT_B_Indx > 0)
					WIRE_Param_Set[1].pVect = &VectorStateMach[m->pCfg->HeadCfg.WP.VECT_B_Indx];
				else
					WIRE_Param_Set[1].pVect = 0;

				if(m->pCfg->HeadCfg.WP.VECT_A_Indx != m->pCfg->HeadCfg.WP.VECT_B_Indx){

					if(m->pCfg->HeadCfg.WP.VECT_A_Indx > 0)
						VectorStateMach[m->pCfg->HeadCfg.WP.VECT_A_Indx].InVal = 0.0;
				}

			}

			//OSC
			Process[m->pCfg->HeadCfg.OSC.PROC_Indx].Param[1] = 0; // Select Calibration
			OSC_TML_Param_Set[0].pVect = &VectorStateMach[m->pCfg->HeadCfg.OSC.VECT_A_Indx];

			if (m->pCfg->HeadCfg.OSC.VECT_A_Indx != m->pCfg->HeadCfg.OSC.VECT_B_Indx)
				VectorStateMach[m->pCfg->HeadCfg.OSC.VECT_B_Indx].Mode = vectSt_Mode_Idle;

			//  AVC
			if (m->pCfg->HeadCfg.AVC.VECT_A_Indx != m->pCfg->HeadCfg.AVC.VECT_B_Indx)
				VectorStateMach[m->pCfg->HeadCfg.AVC.VECT_B_Indx].Mode = vectSt_Mode_Idle;

			switch(curCalib->GenSetup[SETUP_HEAD_SETUP]){

				case BPV_v2_MPGH:
				case BPV_v2_MPGV:
				case BPV_v2_MT_BO_TOS:
				case BPV_v2_TT_BO_TOS:

					VectorStateMach[m->pCfg->HeadCfg.TVL.VECT_Indx].OutVect.softLimits[0] =
					curCalib->Points[CALIB_OSC_SFT_LIMIT].val[0];
					VectorStateMach[m->pCfg->HeadCfg.TVL.VECT_Indx].OutVect.softLimits[1] =
					curCalib->Points[CALIB_OSC_SFT_LIMIT].val[1];

					VectorStateMach[m->pCfg->HeadCfg.OSC.VECT_A_Indx].OutVect.softLimits[0] =
					defCalib->Points[CALIB_OSC_SFT_LIMIT].val[0];
					VectorStateMach[m->pCfg->HeadCfg.OSC.VECT_A_Indx].OutVect.softLimits[1] =
					defCalib->Points[CALIB_OSC_SFT_LIMIT].val[1];

				break;

				default:

					VectorStateMach[m->pCfg->HeadCfg.OSC.VECT_A_Indx].OutVect.softLimits[0] =
					curCalib->Points[CALIB_OSC_SFT_LIMIT].val[0];
					VectorStateMach[m->pCfg->HeadCfg.OSC.VECT_A_Indx].OutVect.softLimits[1] =
					curCalib->Points[CALIB_OSC_SFT_LIMIT].val[1];

				break;

			}

			//AVC
			AVC_Param_Set[0].pVect = &VectorStateMach[m->pCfg->HeadCfg.AVC.VECT_A_Indx];

			if (m->pCfg->HeadCfg.AVC.VECT_A_Indx != m->pCfg->HeadCfg.AVC.VECT_B_Indx)
				VectorStateMach[m->pCfg->HeadCfg.AVC.VECT_B_Indx].Mode = vectSt_Mode_Idle;

			/*
			if(m->pCfg->HeadCfg.EvalateTVLservo_outputs){

				if(TML_MTR_INST[TML_AX_TVL].DigOut_stat[0]){

					if(VectorStateMach[m->pCfg->HeadCfg.TVL.VECT_Indx].xCMD == 0){

						VectorStateMach[m->pCfg->HeadCfg.TVL.VECT_Indx].xCMD = VECT_Set_OUT0;
						//_ToolHeadID 		= m->ToolHeadID;

					}

				}
			}
			*/
			////////////////////////
			if(m->pCfg->HeadCfg.SwitchHead.VECT_Indx > 0 ){

				if(m->pCfg->HeadCfg.SwitchHead.TML_Indx > 0 ){

					if(TML_MTR_INST[m->pCfg->HeadCfg.SwitchHead.TML_Indx -1].DigOut_stat[0]){
					//if(_ToolHeadID_Sw1 != m->ToolHeadID){

						if(VectorStateMach[m->pCfg->HeadCfg.SwitchHead.VECT_Indx-1].xCMD == 0){

							VectorStateMach[m->pCfg->HeadCfg.SwitchHead.VECT_Indx-1].xCMD = VECT_Set_OUT0;
							//_ToolHeadID_Sw1 		= m->ToolHeadID;

						}

					}
				}
			}

			/*
			if(m->pCfg->HeadCfg.SwitchHead.VECT_Indx_2 > 0 ){

				if(m->pCfg->HeadCfg.SwitchHead.VECT_Indx_2 > 0 ){

					if(TML_MTR_INST[m->pCfg->HeadCfg.SwitchHead.TML_Indx_2 -1].DigOut_stat[0]){
					//if(_ToolHeadID_Sw2 != m->ToolHeadID){

						if(VectorStateMach[m->pCfg->HeadCfg.SwitchHead.VECT_Indx_2-1].xCMD == 0){

							VectorStateMach[m->pCfg->HeadCfg.SwitchHead.VECT_Indx_2-1].xCMD = VECT_Set_OUT0;
							//_ToolHeadID_Sw2 		= m->ToolHeadID;
							//_ToolHeadID 		= m->ToolHeadID;

						}

					}
				}
			}
			*/
			/////////////////////

		}

		// REV Direction  - Head A	m->ToolHeadID = 0
		else
		{

			Hardware[1].Outp[5] = 0;	// Select B Head Signal
			Hardware[1].Outp[0] = 0;	// Weld Angle

			//TVL
			Process[m->pCfg->HeadCfg.TVL.PROC_Indx].Param[1] = 0x1 + 0x2; // Select Calibration & Direction

			if(curCalib->GenSetup[SETUP_WF_WP_SWAP] == 0){

				//WF
				Process[m->pCfg->HeadCfg.WF.PROC_Indx].Param[1] = 1; // Select Calibration

				if(m->pCfg->HeadCfg.WF.VECT_B_Indx > 0)
					WIRE_Param_Set[0].pVect = &VectorStateMach[m->pCfg->HeadCfg.WF.VECT_B_Indx];
				else
					WIRE_Param_Set[0].pVect = 0;

				if(m->pCfg->HeadCfg.WF.VECT_A_Indx != m->pCfg->HeadCfg.WF.VECT_B_Indx){

					if(m->pCfg->HeadCfg.WF.VECT_A_Indx > 0)
						VectorStateMach[m->pCfg->HeadCfg.WF.VECT_A_Indx].InVal = 0.0;
				}

				if(m->pCfg->HeadCfg.WF.VECT_Aux_B_Indx > 0)
					WIRE_Param_Set[0].pAuxVect = &VectorStateMach[m->pCfg->HeadCfg.WF.VECT_Aux_B_Indx];
				else
					WIRE_Param_Set[0].pAuxVect = 0;

				if(m->pCfg->HeadCfg.WF.VECT_Aux_A_Indx != m->pCfg->HeadCfg.WF.VECT_Aux_B_Indx){

					if(m->pCfg->HeadCfg.WF.VECT_Aux_A_Indx > 0)
						VectorStateMach[m->pCfg->HeadCfg.WF.VECT_Aux_A_Indx].InVal = 0.0;

				}

				//WP
				Process[m->pCfg->HeadCfg.WP.PROC_Indx].Param[1] = 1; // Select Calibration

				if(m->pCfg->HeadCfg.WP.VECT_B_Indx > 0)
					WIRE_Param_Set[1].pVect = &VectorStateMach[m->pCfg->HeadCfg.WP.VECT_B_Indx];
				else
					WIRE_Param_Set[1].pVect = 0;

				if(m->pCfg->HeadCfg.WP.VECT_A_Indx != m->pCfg->HeadCfg.WP.VECT_B_Indx){

					if(m->pCfg->HeadCfg.WP.VECT_A_Indx > 0)
						VectorStateMach[m->pCfg->HeadCfg.WP.VECT_A_Indx].InVal = 0.0;
				}

			}
			else{

				//WF
				Process[m->pCfg->HeadCfg.WF.PROC_Indx].Param[1] = 0; // Select Calibration

				if(m->pCfg->HeadCfg.WF.VECT_A_Indx > 0)
					WIRE_Param_Set[0].pVect = &VectorStateMach[m->pCfg->HeadCfg.WF.VECT_A_Indx];
				else
					WIRE_Param_Set[0].pVect = 0;

				if(m->pCfg->HeadCfg.WF.VECT_A_Indx != m->pCfg->HeadCfg.WF.VECT_B_Indx){

					if(m->pCfg->HeadCfg.WF.VECT_B_Indx > 0)
						VectorStateMach[m->pCfg->HeadCfg.WF.VECT_B_Indx].InVal = 0.0;
				}

				if(m->pCfg->HeadCfg.WF.VECT_Aux_A_Indx > 0)
					WIRE_Param_Set[0].pAuxVect = &VectorStateMach[m->pCfg->HeadCfg.WF.VECT_Aux_A_Indx];
				else
					WIRE_Param_Set[0].pAuxVect = 0;

				if(m->pCfg->HeadCfg.WF.VECT_Aux_A_Indx != m->pCfg->HeadCfg.WF.VECT_Aux_B_Indx){

					if(m->pCfg->HeadCfg.WF.VECT_Aux_B_Indx > 0)
						VectorStateMach[m->pCfg->HeadCfg.WF.VECT_Aux_B_Indx].InVal = 0.0;
				}

				//WP
				Process[m->pCfg->HeadCfg.WP.PROC_Indx].Param[1] = 0; // Select Calibration

				if(m->pCfg->HeadCfg.WP.VECT_A_Indx > 0)
					WIRE_Param_Set[1].pVect = &VectorStateMach[m->pCfg->HeadCfg.WP.VECT_A_Indx];
				else
					WIRE_Param_Set[1].pVect = 0;

				if(m->pCfg->HeadCfg.WP.VECT_A_Indx != m->pCfg->HeadCfg.WP.VECT_B_Indx){

					if(m->pCfg->HeadCfg.WP.VECT_B_Indx > 0)
						VectorStateMach[m->pCfg->HeadCfg.WP.VECT_B_Indx].InVal = 0.0;
				}

			}

			//OSC
			Process[m->pCfg->HeadCfg.OSC.PROC_Indx].Param[1] = 1; // Select Calibration
			OSC_TML_Param_Set[0].pVect = &VectorStateMach[m->pCfg->HeadCfg.OSC.VECT_B_Indx];

			if (m->pCfg->HeadCfg.OSC.VECT_A_Indx != m->pCfg->HeadCfg.OSC.VECT_B_Indx)
				VectorStateMach[m->pCfg->HeadCfg.OSC.VECT_A_Indx].Mode = vectSt_Mode_Idle;

			// AVC
			if (m->pCfg->HeadCfg.AVC.VECT_A_Indx != m->pCfg->HeadCfg.AVC.VECT_B_Indx)
				VectorStateMach[m->pCfg->HeadCfg.AVC.VECT_A_Indx].Mode = vectSt_Mode_Idle;

			switch(curCalib->GenSetup[SETUP_HEAD_SETUP]){

				case BPV_v2_MPGH:
				case BPV_v2_MPGV:
				case BPV_v2_MT_BO_TOS:
				case BPV_v2_TT_BO_TOS:

					VectorStateMach[m->pCfg->HeadCfg.TVL.VECT_Indx].OutVect.softLimits[0] =
					curCalib->Points[CALIB_OSC_SFT_LIMIT].val[0];
					VectorStateMach[m->pCfg->HeadCfg.TVL.VECT_Indx].OutVect.softLimits[1] =
					curCalib->Points[CALIB_OSC_SFT_LIMIT].val[1];

					VectorStateMach[m->pCfg->HeadCfg.OSC.VECT_B_Indx].OutVect.softLimits[0] =
					defCalib->Points[CALIB_OSC_SFT_LIMIT].val[2];
					VectorStateMach[m->pCfg->HeadCfg.OSC.VECT_B_Indx].OutVect.softLimits[1] =
					defCalib->Points[CALIB_OSC_SFT_LIMIT].val[3];

				break;

				default:

					VectorStateMach[m->pCfg->HeadCfg.OSC.VECT_B_Indx].OutVect.softLimits[0] =
					curCalib->Points[CALIB_OSC_SFT_LIMIT].val[2];
					VectorStateMach[m->pCfg->HeadCfg.OSC.VECT_B_Indx].OutVect.softLimits[1] =
					curCalib->Points[CALIB_OSC_SFT_LIMIT].val[3];

				break;

			}

			//AVC
			AVC_Param_Set[0].pVect = &VectorStateMach[m->pCfg->HeadCfg.AVC.VECT_B_Indx];

			if (m->pCfg->HeadCfg.AVC.VECT_A_Indx != m->pCfg->HeadCfg.AVC.VECT_B_Indx)
				VectorStateMach[m->pCfg->HeadCfg.AVC.VECT_A_Indx].Mode = vectSt_Mode_Idle;

			/*
			if(m->pCfg->HeadCfg.EvalateTVLservo_outputs){

				if(!TML_MTR_INST[TML_AX_TVL].DigOut_stat[0]){

					if(VectorStateMach[m->pCfg->HeadCfg.TVL.VECT_Indx].xCMD == 0){

						VectorStateMach[m->pCfg->HeadCfg.TVL.VECT_Indx].xCMD = VECT_Rst_OUT0;
						//_ToolHeadID 		= m->ToolHeadID;

					}

				}
			}
			*/
			////////////////////////
			if(m->pCfg->HeadCfg.SwitchHead.VECT_Indx > 0 ){

				if(m->pCfg->HeadCfg.SwitchHead.TML_Indx > 0 ){

					if(!TML_MTR_INST[m->pCfg->HeadCfg.SwitchHead.TML_Indx -1].DigOut_stat[0]){
					//if(_ToolHeadID_Sw1 != m->ToolHeadID){

						if(VectorStateMach[m->pCfg->HeadCfg.SwitchHead.VECT_Indx-1].xCMD == 0){

							VectorStateMach[m->pCfg->HeadCfg.SwitchHead.VECT_Indx-1].xCMD = VECT_Rst_OUT0;
							//_ToolHeadID_Sw1 		= m->ToolHeadID;
							//_ToolHeadID 		= m->ToolHeadID;

						}

					}
				}
			}

			/*
			if(m->pCfg->HeadCfg.SwitchHead.VECT_Indx_2 > 0 ){

				if(m->pCfg->HeadCfg.SwitchHead.TML_Indx_2 > 0 ){

					if(!TML_MTR_INST[m->pCfg->HeadCfg.SwitchHead.TML_Indx_2 -1].DigOut_stat[0]){
					//if(_ToolHeadID_Sw2 != m->ToolHeadID){

						if(VectorStateMach[m->pCfg->HeadCfg.SwitchHead.VECT_Indx_2-1].xCMD == 0){

							VectorStateMach[m->pCfg->HeadCfg.SwitchHead.VECT_Indx_2-1].xCMD = VECT_Rst_OUT0;
							//_ToolHeadID_Sw2 		= m->ToolHeadID;
							//_ToolHeadID 		= m->ToolHeadID;

						}

					}
				}
			}
			*/
			/////////////////////

		}

		if (m->ToolHeadID != _ToolHeadID){
			_ToolHeadID 		= m->ToolHeadID;

			if(m->pCfg->HeadCfg.GEN.Torch_Mode == MODE_DUAL_OSCILATOR)
				Process[m->pCfg->HeadCfg.OSC.PROC_Indx].xCMD = prcsRESTART;

			if(m->pCfg->HeadCfg.GEN.AVC_Mode == MODE_DUAL_AVC)
				Process[m->pCfg->HeadCfg.AVC.PROC_Indx].xCMD = prcsRESTART;

		}

		// On page calibration No limits and Force ToolID assigments
		if (hmi->curHeadID == P_MODE_OSC_LIMIT_CALIB)
		{

			switch(curCalib->GenSetup[SETUP_HEAD_SETUP]){

				case BPV_v2_MPGH:
				case BPV_v2_MPGV:
				case BPV_v2_MT_BO_TOS:
				case BPV_v2_TT_BO_TOS:

					VectorStateMach[m->pCfg->HeadCfg.TVL.VECT_Indx].OutVect.softLimits[0] =
					defCalib->Points[CALIB_OSC_SFT_LIMIT].val[0];
					VectorStateMach[m->pCfg->HeadCfg.TVL.VECT_Indx].OutVect.softLimits[1] =
					defCalib->Points[CALIB_OSC_SFT_LIMIT].val[1];

					VectorStateMach[m->pCfg->HeadCfg.OSC.VECT_A_Indx].OutVect.softLimits[0] =
					defCalib->Points[CALIB_OSC_SFT_LIMIT].val[0];
					VectorStateMach[m->pCfg->HeadCfg.OSC.VECT_A_Indx].OutVect.softLimits[1] =
					defCalib->Points[CALIB_OSC_SFT_LIMIT].val[1];

					VectorStateMach[m->pCfg->HeadCfg.OSC.VECT_B_Indx].OutVect.softLimits[0] =
					defCalib->Points[CALIB_OSC_SFT_LIMIT].val[2];
					VectorStateMach[m->pCfg->HeadCfg.OSC.VECT_B_Indx].OutVect.softLimits[1] =
					defCalib->Points[CALIB_OSC_SFT_LIMIT].val[3];

				break;

				default:

					VectorStateMach[m->pCfg->HeadCfg.OSC.VECT_A_Indx].OutVect.softLimits[0] =
					defCalib->Points[CALIB_OSC_SFT_LIMIT].val[0];
					VectorStateMach[m->pCfg->HeadCfg.OSC.VECT_A_Indx].OutVect.softLimits[1] =
					defCalib->Points[CALIB_OSC_SFT_LIMIT].val[1];

					VectorStateMach[m->pCfg->HeadCfg.OSC.VECT_B_Indx].OutVect.softLimits[0] =
					defCalib->Points[CALIB_OSC_SFT_LIMIT].val[2];
					VectorStateMach[m->pCfg->HeadCfg.OSC.VECT_B_Indx].OutVect.softLimits[1] =
					defCalib->Points[CALIB_OSC_SFT_LIMIT].val[3];

				break;

			}

		}

		///////////////////////////////////////////////////////////////
		FinalPos			= StartPos + (DINT)curCfg->Param[parTVL_RunDist].val[0];

		//////////

		/*#ifdef MIG_PENDANT

		//intrf->GlblBtnCmd[0] = (HMI_Intr.GlblBtnCmd[0] & 0xFFFFFFFE);

			intrf->_intr._GlblBtnCmd[0] = (HMI_Intr.GlblBtnCmd[0] & (0xFFFFFFFF - ANDR_BTN_HOME)) ;
			intrf->_intr._GlblBtnCmd[1] = HMI_Intr.GlblBtnCmd[1];

		#else*/

			intrf->_intr._GlblBtnCmd[0] = (intrf->GlblBtnCmd[0] & (0xFFFFFFFF - ANDR_BTN_HOME)) ;
			intrf->_intr._GlblBtnCmd[1] = intrf->GlblBtnCmd[1];

		//#endif

		// THIS MUST BE RUN //
		// This is for pipe compensation

		if(m->FrameDia > 0.0)
			curCalib->GenFloatValue[SETUP_FLOAT_TRACK_DIA] = m->FrameDia ;

		if(hmi->curHeadID != P_MODE_TVL_CALIB){

			if(WRST_TML_Param_Set[0].MappingActive > 0)
				TVL_ROT_Param_Set[0].TotalRescaleFactor = WRST_TML_Param_Set[0].TVLSpeedOverride;

			else if((curCfg->Param[parTVL_TrackDia].val[0]> 0.0) && (curCalib->GenFloatValue[SETUP_FLOAT_TRACK_DIA]> 0.0))
				TVL_ROT_Param_Set[0].TotalRescaleFactor = curCfg->Param[parTVL_TrackDia].val[0] / curCalib->GenFloatValue[SETUP_FLOAT_TRACK_DIA];

			else
				TVL_ROT_Param_Set[0].TotalRescaleFactor = 1.0;

		}
		else
			TVL_ROT_Param_Set[0].TotalRescaleFactor = 1.0;

		sm_serv(&m->sm);
		TimerExecute(&ESTOP_Dly_Tmr);
		TimerExecute(&DoubleStop_TMR);
		LoggerSrv(&LogMgr);

		//AndroidHelper(m , 0);
		SetBannerTxt(m, hmi, intrf);
		TimerExecute(&AndroidConnect_Tmr);

		RestartStateMach();

		_datagramCountTotal[0] = datagramCountTotal[0];
		_datagramPerSec[0]	= datagramPerSec[0];

		if (btnProgress < btnProgressMax)
			btnProgress++;

		KK_Life++;

		/////////////////////////////////////////////////////

		LastHeadDir = (USINT)Master[0].ToolHeadID;

		if(Ready2StoreLastPos){

			// Store last Position
			if (TML_MTR_INST[m->pCfg->HeadCfg.OSC.TML_A_Indx]._int.Init &&
				 (TML_MTR_INST[m->pCfg->HeadCfg.OSC.TML_A_Indx]._cfg.absFbk != 2))
				OLD_MTR_POS[OSC_LAST_POS] = AxisCh[m->pCfg->HeadCfg.OSC.TML_A_Indx].curPos;

			if (TML_MTR_INST[m->pCfg->HeadCfg.WRST.TML_A_Indx]._int.Init &&
				 (TML_MTR_INST[m->pCfg->HeadCfg.WRST.TML_A_Indx]._cfg.absFbk != 2))
				OLD_MTR_POS[WRST_LAST_POS] = AxisCh[m->pCfg->HeadCfg.WRST.TML_A_Indx].curPos;

			if (TML_MTR_INST[m->pCfg->HeadCfg.TVL.TML_Indx]._int.Init &&
				 (TML_MTR_INST[m->pCfg->HeadCfg.TVL.TML_Indx]._cfg.absFbk != 2))
				OLD_MTR_POS[TVL_LAST_POS] = AxisCh[m->pCfg->HeadCfg.TVL.TML_Indx].curPos;

			switch(curCalib->GenSetup[SETUP_HEAD_SETUP]){

				case CLAMSHELL_HEAD:
				case CHERRYPOINT_BP1_HEAD:
				case CHERRYPOINT_BP2_HEAD:
				case CHERRYPOINT_MT_BP2_HEAD:
				case MIG_TIG_HEAD:
				case BPV_F_HEAD:
				//dodane 6Dec23
				case BPV_v1_MT:

					OLD_MTR_POS[INDX_A_LAST_POS] = DC_Mtr[m->pCfg->HeadCfg.INDX.DC_A_Indx].msc.Pos;
					OLD_MTR_POS[INDX_B_LAST_POS] = DC_Mtr[m->pCfg->HeadCfg.INDX.DC_B_Indx].msc.Pos;

					//curCalib->GenSetup[SETUP_MAPPING_ON] = MAPPING_OFF;
					//WRST_TML_Param_Set[0].MappingActive = 0;

				break;

				case BPV_v2:
				case BPV_v2_MPBO:
				case BPV_v2_MPGH:
				case BPV_v2_MPGV:
				// dodane 8July24
				case BPV_v2_Video:
				//dodane 6Dec23
				case BPV_v2_MT:

					if (TML_MTR_INST[m->pCfg->HeadCfg.INDX.TML_A_Indx]._int.Init &&
						(TML_MTR_INST[m->pCfg->HeadCfg.INDX.TML_A_Indx]._cfg.absFbk != 2))
						OLD_MTR_POS[INDX_A_LAST_POS] = AxisCh[m->pCfg->HeadCfg.INDX.TML_A_Indx].curPos;

					if (TML_MTR_INST[m->pCfg->HeadCfg.INDX.TML_B_Indx]._int.Init &&
						(TML_MTR_INST[m->pCfg->HeadCfg.INDX.TML_B_Indx]._cfg.absFbk != 2))
						OLD_MTR_POS[INDX_B_LAST_POS] = AxisCh[m->pCfg->HeadCfg.INDX.TML_B_Indx].curPos;

				break;

				default:

				break;

			}

		}

		//////////
		if(m->WireDisabled != _WireDisabled)
			LogTxt(&LogMgr, "Wire Disable Change %d" , (DINT)m->WireDisabled);

		_WireDisabled = m->WireDisabled;

	}

	/*********************************************************/
	/****	Process parameters assigments	************************/
	DINT MasterSequence(MASTER_typ * m, HMI_typ * hmi, plcbit StartBtn, plcbit StopBtn)
	{
	int 			i;
	char			status;
	DINT			ret;
	DINT			d;
	USINT			newFile;

	//Cfg_typ *cfg;
	CurCfg_typ *	curCfg;

	//CurCalib_typ *curCalib , *defCalib;
	//Scaled_Var_obj *var;
	//cfg = (Cfg_typ*) m->pCfg;
	curCfg				= (CurCfg_typ *)
	m->pCurCfg;

	//curCalib = (CurCalib_typ*) m->pCalib;
	//defCalib = (CurCalib_typ*) m->pDefaultCalib;
	//var = (Scaled_Var_obj*) m->pScaledVar;
	m->TestMode 		= intrf->TestMode;

	ret 				= 0;

	if((hmi->curHeadID == 0xFFFE)){ // Screen RUn or Alter Run

		if(intrf->GlblBtnCmd[0] &ANDR_BTN_UP){

			AVC_Param_Set[0].BoostCmd = 1;
			PS_Param_Set[0].BoostCmd = 1;
			TVL_ROT_Param_Set[0].BoostCmd = 1;
			WIRE_Param_Set[0].BoostCmd = 1;
			WIRE_Param_Set[1].BoostCmd = 1;

		}
		else if(intrf->GlblBtnCmd[0] &ANDR_BTN_DOWN){

			AVC_Param_Set[0].BoostCmd = 2;
			PS_Param_Set[0].BoostCmd = 2;
			TVL_ROT_Param_Set[0].BoostCmd = 2;
			WIRE_Param_Set[0].BoostCmd = 2;
			WIRE_Param_Set[1].BoostCmd = 2;

		}
		else{

			AVC_Param_Set[0].BoostCmd = 0;
			PS_Param_Set[0].BoostCmd = 0;
			TVL_ROT_Param_Set[0].BoostCmd = 0;
			WIRE_Param_Set[0].BoostCmd = 0;
			WIRE_Param_Set[1].BoostCmd = 0;

		}
	}
	else{

		AVC_Param_Set[0].BoostCmd = 0;
		PS_Param_Set[0].BoostCmd = 0;
		TVL_ROT_Param_Set[0].BoostCmd = 0;
		WIRE_Param_Set[0].BoostCmd = 0;
		WIRE_Param_Set[1].BoostCmd = 0;

	}

	/////////
	if (StopBtn)
	{
		AutoStartBtn		= 0;

		if (TimerIsTimeOut(&DoubleStop_TMR))
			TimerStart(&DoubleStop_TMR, 0.5);
		else
			DoubleStopBtn_Latch = 1;
	}

	if (StopBtn)
		StopBtn_Latch = 1;

	if (Process[m->pCfg->HeadCfg.TVL.PROC_Indx].Status != prcsSTATUS_Stopped)
	{
		if(m->SubSeqStep == 1 )// Weld to Target
		{
			if(abs(m->curSegm[ACT_TVL_DIST] - Process[m->pCfg->HeadCfg.TVL.PROC_Indx].Param[0]) < 10)
				m->SubSeqStep = 2;
		}
	}

	if ((Process[m->pCfg->HeadCfg.TVL.PROC_Indx].Status == prcsSTATUS_Stopped) ||
	(Process[m->pCfg->HeadCfg.TVL.PROC_Indx].Status == prcsSTATUS_ReturnDly)){

		if (DoubleStopBtn_Latch)
			m->SubSeqStep = 0;
	}
	DoubleStopBtn_Latch = 0;

	if(curCfg->Param_ENUM[parENUM_TVL_MODE].val[0] == 3) // Continues welding
		m->SubSeqStep = 0;

	if (StopBtn_Latch)
		Process[m->pCfg->HeadCfg.TVL.PROC_Indx].Param[2] = 0; // No Auto Stop and Not Rewrap

	//////////////////////////
	////////////////////////////
	if (m->SeqStep > 0)
		GlobalTimer += 0.0512; // Timer based on task class

	//////////////

		//	 MASTER SEQUENCE  //
	switch (m->SeqStep)
	{
		case 0:

			//////////////////////////////////////
			if(curCfg->Param[parGEN_WeldProgramRepeat].val[0] == 0.0)
				File_RW._int.PathDoneCnt = 0;

			// Reset Disable when was in Test Mode
			Process[m->pCfg->HeadCfg.AVC.PROC_Indx].Disable &= 0xFD;
			Process[m->pCfg->HeadCfg.OSC.PROC_Indx].Disable &= 0xFD;
			Process[m->pCfg->HeadCfg.TVL.PROC_Indx].Disable &= 0xFD;
			Process[m->pCfg->HeadCfg.TIG.PROC_Indx].Disable &= 0xFD;
			Process[m->pCfg->HeadCfg.HW.PROC_Indx].Disable &= 0xFD;
			StopBtn_Latch = 0;

			// AVC Locked is OFF

			//if(curCfg->Param_ENUM[parENUM_AVC_Mode].val[0] != 3) // AVC Mode NOT LOCKED !
				//Process[m->pCfg->HeadCfg.AVC.PROC_Indx].Param[0] = 0;

			if(StartBtn && !Check_OSC_Amplt_and_Center())
				break;

			if (StopBtn)
			{
				LogTxt(&LogMgr, "Quick stop");
				m->SeqStep = 254;			// Halt Stop
				break;
			}

			status = 1;

			if (//(Process[m->pCfg->HeadCfg.GAS.PROC_Indx].Status != prcsSTATUS_Stopped)
				(Process[m->pCfg->HeadCfg.AVC.PROC_Indx].Status != prcsSTATUS_Stopped) ||
				(Process[m->pCfg->HeadCfg.OSC.PROC_Indx].Status != prcsSTATUS_Stopped) ||
				(Process[m->pCfg->HeadCfg.TVL.PROC_Indx].Status != prcsSTATUS_Stopped) ||
				(Process[m->pCfg->HeadCfg.WF.PROC_Indx].Status != prcsSTATUS_Stopped))
				//(Process[m->pCfg->HeadCfg.WP.PROC_Indx].Status != prcsSTATUS_Stopped))
				status = 0;

			if (status)
			{

				if (!ErrorMgr.Error)
				{
					ret = 1;		// Raedy To Run

					if((intrf->GlblBtnCmd[0] &ANDR_BTN_HOME) && StartBtn){

						Process[m->pCfg->HeadCfg.TVL.PROC_Indx].Param[3] = 0;
						Process[m->pCfg->HeadCfg.TVL.PROC_Indx].Param[2] = 2; //only rewrap
						Process[m->pCfg->HeadCfg.TVL.PROC_Indx].xCMD = prcsSTART;
						m->SeqStep = 210;

					}

					//if ((StartBtn || AutoStartBtn) && (XMLHelper.xCmd != XML_CMD_READ))
					//else if ((StartBtn || AutoStartBtn) && ((Weld_Report_Status < 2) || ((curCalib->GenSetup[SETUP_EXTRAS]&0x1) == 0))) //Weld_Report_Mode
					else if ((StartBtn || AutoStartBtn) && ((Weld_Report_Start_Enable) || ((curCalib->GenSetup[SETUP_EXTRAS]&0x1) == 0))) //Weld_Report_Mode
					{
						Weld_Report_Status = 1;

						AutoStartBtn = 0;

						if (m->SubSeqStep == 2)
						{ // Rewrap

							if (curCalib->GenSetup[SETUP_SOUND_DELAY] || curCalib->GenSetup[SETUP_AUTO_START])
								TimerStart(&m->sm.Tmr1, curCalib->GenFloatValue[SETUP_FLOAT_SOUND_TM]);

							else
								TimerStart(&m->sm.Tmr1, 0.1);

							m->SeqStep = 150;

						}
						else
						{

						GlobalTimer 		= 0;

						LogTxt(&LogMgr, "PreProcess start");

						if (curCalib->GenSetup[SETUP_SOUND_DELAY] || curCalib->GenSetup[SETUP_AUTO_START])
							TimerStart(&m->sm.Tmr1, curCalib->GenFloatValue[SETUP_FLOAT_SOUND_TM]);
						else
							TimerStart(&m->sm.Tmr1, 0.1);

							m->SeqStep++;

						}
					}

					/*
					else if ((StartBtn || AutoStartBtn) && (XMLHelper.xCmd == XML_CMD_READ)){

						strcpy(hmi->pMessage[0], " FILE OPER. \n ");
						strcpy(hmi->pMessage[1], File_RW.fileName);
						strcpy(hmi->pMessage[2], "Is Loading");
						strcpy(hmi->pMessage[3] ,"Wait for finish");

						Set_Message(hmi , 0.1);

					}
					*/
				}

			}
			else
			{
				if (StopBtn)
				{
					LogTxt(&LogMgr, "Some Prcs aborted");
					m->SeqStep = 254;
				}

			}

		break;

		case 1:
		// Always Coolant On
			if (!m->TestMode)
			{
				if (Process[m->pCfg->HeadCfg.COOL.PROC_Indx].Status != prcsSTATUS_Run)
					Process[m->pCfg->HeadCfg.COOL.PROC_Indx].xCMD = prcsSTART;
			}

			ret = 2; // Preparig To Run

			if (StopBtn)
			{
				LogTxt(&LogMgr, "Some Prcs aborted");
				m->SeqStep = 254;
			}
			else if (ErrorMgr.Error)
				m->SeqStep = 100;

			else if (!TimerIsTimeOut(&m->sm.Tmr1))
				break;

			else
			{
				if (!m->TestMode)
				{
					Process[m->pCfg->HeadCfg.GAS.PROC_Indx].xCMD = prcsSTART;
					Process[m->pCfg->HeadCfg.COOL.PROC_Indx].xCMD = prcsSTART;
				}

				if (m->TestMode)
				{

					//Process[m->pCfg->HeadCfg.AVC.PROC_Indx].Disable |= 0x02 ;
					Process[m->pCfg->HeadCfg.AVC.PROC_Indx].TestMode = 1;
					Process[m->pCfg->HeadCfg.TIG.PROC_Indx].Disable |= 0x02;
					Process[m->pCfg->HeadCfg.HW.PROC_Indx].Disable |= 0x02;

				}
				else
				{

					if ((Process[m->pCfg->HeadCfg.GAS.PROC_Indx].Status == prcsSTATUS_Run) &&
					(Process[m->pCfg->HeadCfg.COOL.PROC_Indx].Status == prcsSTATUS_Run))
					{
						//Process[m->pCfg->HeadCfg.AVC.PROC_Indx].Disable &= 0xFD ;
						Process[m->pCfg->HeadCfg.AVC.PROC_Indx].TestMode = 0;
						Process[m->pCfg->HeadCfg.TIG.PROC_Indx].Disable &= 0xFD;
						Process[m->pCfg->HeadCfg.HW.PROC_Indx].Disable &= 0xFD;

					}
					else
						break;

				}

				Process[m->pCfg->HeadCfg.AVC.PROC_Indx].xCMD = prcsSTART;

				//if(!m->TestMode)
				Process[m->pCfg->HeadCfg.TIG.PROC_Indx].xCMD = prcsForceON;

				LogTxt(&LogMgr, "ARC start");

				m->SeqStep++;

			}

		break;

		case 2:

			// Always Coolant On
			if (!m->TestMode)
			{
				if (Process[m->pCfg->HeadCfg.COOL.PROC_Indx].Status != prcsSTATUS_Run)
					Process[m->pCfg->HeadCfg.COOL.PROC_Indx].xCMD = prcsSTART;
			}

			ret = 2; // Preparig To Run

			if (StopBtn)
			{
				LogTxt(&LogMgr, "Some Prcs aborted");
				m->SeqStep			= 254;
			}

			///////////////////////////
			else if (ErrorMgr.Error)
				m->SeqStep = 100;

			else if ((Process[m->pCfg->HeadCfg.AVC.PROC_Indx].Status == prcsSTATUS_Run)
					|| (Process[m->pCfg->HeadCfg.AVC.PROC_Indx].Status == prcsSTATUS_AVC_OK))
			{

				Process[m->pCfg->HeadCfg.OSC.PROC_Indx].xCMD = prcsSTART;
				Process[m->pCfg->HeadCfg.OSC.PROC_Indx].Param[0] = 0; // Start with ramp
				Process[m->pCfg->HeadCfg.TIG.PROC_Indx].xCMD = prcsSTART;

				/*	TVL */
				Process[m->pCfg->HeadCfg.TVL.PROC_Indx].Param[2] = m->SubSeqStep;
				Process[m->pCfg->HeadCfg.TVL.PROC_Indx].xCMD = prcsSTART;

#ifdef EXTENDED_LOGS
				LogTxt(&LogMgr, "M:TVL%d Start: %.2f" , (UDINT) m->ToolHeadID , ABS_TVL_Pos);
#endif
				StartPos = 0;

				CalculateRunOverlap();

				if (!m->WireDisabled)
				{
					// if prcsStart then Param[0] = 0 is set in Wire process - jus in case
					//Process[m->pCfg->HeadCfg.WF.PROC_Indx].Param[0] = 0; // start with full ramp
					Process[m->pCfg->HeadCfg.WF.PROC_Indx].xCMD = prcsSTART;
					//Process[m->pCfg->HeadCfg.WP.PROC_Indx].Param[0] = 0; // start with full ramp
					Process[m->pCfg->HeadCfg.WP.PROC_Indx].xCMD = prcsSTART;
					Process[m->pCfg->HeadCfg.HW.PROC_Indx].xCMD = prcsSTART;
				}

				LogTxt(&LogMgr, "ARC established");

				TimerStart(&WireDisable_TMR, 3.0);

				m->SeqStep++;

			}

		break;

		case 3:
			// Always Coolant On
			if (!m->TestMode)
			{
				if (Process[m->pCfg->HeadCfg.COOL.PROC_Indx].Status != prcsSTATUS_Run)
					Process[m->pCfg->HeadCfg.COOL.PROC_Indx].xCMD = prcsSTART;
			}

			WireDisableInable(WireDisable_TMR.Q);
			Process[m->pCfg->HeadCfg.TIG.PROC_Indx].Param[0] = Process[m->pCfg->HeadCfg.OSC.PROC_Indx].subStatus;
			Process[m->pCfg->HeadCfg.HW.PROC_Indx].Param[0] = Process[m->pCfg->HeadCfg.OSC.PROC_Indx].subStatus;
			ret = 3; //  Run

			if (curCfg->Param_ENUM[parENUM_WeldProgramLinkMode].val[0] > 0.0)
			{

				if(curCfg->Param[parGEN_WeldProgramRepeat].val[0] == 0.0)
				{

					if (strlen(curCfg->NextProgramName) > 0)
					{

						if (!strstr(curCfg->NextProgramName, "NONE"))
						{ // Not None

							// It should be some additional condition when to load new file
							if (actRot != _actRot){
								//TakeNextWeldProgram(hmi);
								//newFile 			= 1;

							}

						}

					}

				}

			}

			_actRot = actRot;

			if (Process[m->pCfg->HeadCfg.TVL.PROC_Indx].subStatus == 1)
			{ // End of travel reached
				//LogTxt(&LogMgr, "Path Done");
				//LogTxt(&LogMgr, "Path Done: %.2f" , ABS_TVL_Pos);
				Weld_Report_Status = 2;
				m->SeqStep = 200;
			}

			if (StopBtn)
			{
				LogTxt(&LogMgr, "Process stop");
				//Process[m->pCfg->HeadCfg.TVL.PROC_Indx].xCMD = prcsSTOP;
				m->SeqStep = 200;

			}
			else if (ErrorMgr.Error || m->ESTOP)
			{
				LogTxt(&LogMgr, "Process Error");
				m->SeqStep = 100;
			}

		break;

		case 100:
			// Always Coolant On
			if (!m->TestMode)
			{
				if (Process[m->pCfg->HeadCfg.COOL.PROC_Indx].Status != prcsSTATUS_Run)
					Process[m->pCfg->HeadCfg.COOL.PROC_Indx].xCMD = prcsSTART;
			}

			Process[m->pCfg->HeadCfg.TVL.PROC_Indx].xCMD = prcsHalt;
			Process[m->pCfg->HeadCfg.OSC.PROC_Indx].xCMD = prcsHalt;
			Process[m->pCfg->HeadCfg.AVC.PROC_Indx].xCMD = prcsHalt;
			Process[m->pCfg->HeadCfg.WF.PROC_Indx].xCMD = prcsHalt;
			Process[m->pCfg->HeadCfg.WP.PROC_Indx].xCMD = prcsHalt;
			Process[m->pCfg->HeadCfg.TIG.PROC_Indx].xCMD = prcsHalt;
			Process[m->pCfg->HeadCfg.HW.PROC_Indx].xCMD = prcsHalt;
			Process[m->pCfg->HeadCfg.GAS.PROC_Indx].xCMD = prcsSTOP;

			//Process[m->pCfg->HeadCfg.COOL.PROC_Indx].xCMD = prcsHalt;
			switch (ErrorMgr.Error)
			{
				case ERROR_FATAL:
					m->SeqStep++;
				break;

				case ERROR_MOTOR:
					m->SeqStep++;
				break;

				case ERROR_MOTOR_INIT:
					m->SeqStep++;
				break;

				case ERROR_TIG_PROC:
					m->SeqStep++;
				break;

				default:
					m->SeqStep++;
				break;
			}

		break;

		case 101:
			ret = 4; // Preparig To Stop in Halt Mode

			if (StopBtn)
			{
				for (i = 0; i < PROCESS_NUM; i++)
				{
					if (i != PROC_COOL)
						Process[i].xCMD = prcsHalt;
				}
				Process[m->pCfg->HeadCfg.GAS.PROC_Indx].xCMD = prcsSTOP; // maintain gas
			}

			status = 1;

			if (Process[m->pCfg->HeadCfg.TVL.PROC_Indx].Status != prcsSTATUS_Stopped)
				status = 0;

			if (Process[m->pCfg->HeadCfg.OSC.PROC_Indx].Status != prcsSTATUS_Stopped)
				status = 0;

			if (Process[m->pCfg->HeadCfg.AVC.PROC_Indx].Status != prcsSTATUS_Stopped)
				status = 0;

			if (Process[m->pCfg->HeadCfg.WF.PROC_Indx].Status != prcsSTATUS_Stopped)
				status = 0;

			if (Process[m->pCfg->HeadCfg.GAS.PROC_Indx].Status != prcsSTATUS_Stopped)
				status = 0;

			if (Process[m->pCfg->HeadCfg.WP.PROC_Indx].Status != prcsSTATUS_Stopped)
				status = 0;

			if (Process[m->pCfg->HeadCfg.TIG.PROC_Indx].Status != prcsSTATUS_Stopped)
				status = 0;

			if (Process[m->pCfg->HeadCfg.HW.PROC_Indx].Status != prcsSTATUS_Stopped)
				status = 0;

			if (status)
			{
				LogTxt(&LogMgr, "Prc Final stopped");
				m->SeqStep = 254;
			}

		break;

		case 150:

			if (StopBtn)
			{
				LogTxt(&LogMgr, "Quick stop");
				m->SeqStep = 254;			// Quick Stop
				break;
			}

			if (!TimerIsTimeOut(&m->sm.Tmr1))
				break;

			/*	TVL */
			Process[m->pCfg->HeadCfg.TVL.PROC_Indx].Param[2] = m->SubSeqStep;
			Process[m->pCfg->HeadCfg.TVL.PROC_Indx].xCMD = prcsSTART;
			StartPos = 0;

			CalculateRunOverlap();

			m->SeqStep = 202;

		break;

		case 200:

			// Always Coolant On
			if (!m->TestMode)
			{
				if (Process[m->pCfg->HeadCfg.COOL.PROC_Indx].Status != prcsSTATUS_Run)
					Process[m->pCfg->HeadCfg.COOL.PROC_Indx].xCMD = prcsSTART;
			}

			for (i = 0; i < PROCESS_NUM; i++)
			{
				if ((i != PROC_COOL)) //&&( i != m->pCfg->HeadCfg.TVL.PROC_Indx))
					Process[i].xCMD = prcsSTOP;

			}

			/*
			if(CurCalib.GenSetup[SETUP_CONTIN_WELD] != 0){ // Not Standard Mode
			//if(CurCfg.Param_ENUM[parENUM_TVL_MODE].val[0] != 3){ // NOT Continues welding
```
